PROGRAM F60_METS_Outputs
VAR
	//test : BOOL;
	fbForceOutputs					: FB_IO2_ForceOutputs;

	fbEUCAMachineRun_PulseGen		: FB_SquareWave;
	fbCaseContentOK_PulseGen		: FB_SquareWave;
	fbCaseValidationOK_PulseGen		: FB_SquareWave;
	fbOuterValidationOK_PulseGen	: FB_SquareWave;
	fbLabellerInhibit_PulseGen			: FB_SquareWave;
	fbTPDMachineRun_PulseGen		: FB_SquareWave;


	fbSafetyResetSignal				: FB_IO2_OutputCtrl;		(**)
	fbAdditionalSafetyResetSignal		: FB_IO2_OutputCtrl;
	fbResetPBIndicator					: FB_IO2_OutputCtrl;

	tofTPDMachineRunOff				: TOF;
	tofEUCAPreMachineRunOff			: TOF;
	tofEUCAMachineRunOff			: TOF;

	fbTPDMachineRun				: FB_IO2_OutputCtrl;
	fbCMLConvoyerRun			: FB_IO2_OutputCtrl;
	fbEUCAPreMachineRun			: FB_IO2_OutputCtrl;
	fbEUCAMachineRun			: FB_IO2_OutputCtrl;

	fbCaseContentOK				: FB_IO2_OutputCtrl;
	fbCaseValidationOK			: FB_IO2_OutputCtrl;
	fbOuterValidationOK			: FB_IO2_OutputCtrl;
	fbLabellerInhibit				: FB_IO2_OutputCtrl;

	ftrigPrintWhiteLable			: F_TRIG;

	fbPackAggregCamLensAir		: FB_IO2_OutputCtrl;
	fbOuterAggregCamLensAir	: FB_IO2_OutputCtrl;

	(*fbMLCameraLightning			: FB_IO2_OutputCtrl;
	fbAggCameraLightning		: FB_IO2_OutputCtrl;
	fbConfCameraLightning		: FB_IO2_OutputCtrl;
	fbOuterAggCameraLightning	: FB_IO2_OutputCtrl;*

	fbCamera01Lightning				: FB_IO2_OutputCtrl;
	fbCamera02Lightning				: FB_IO2_OutputCtrl;
	fbCamera03Lightning				: FB_IO2_OutputCtrl;
	fbCamera04Lightning				: FB_IO2_OutputCtrl;
	fbCamera05Lightning				: FB_IO2_OutputCtrl;
	fbCamera06Lightning				: FB_IO2_OutputCtrl;
	fbCamera07Lightning				: FB_IO2_OutputCtrl;
	fbCamera08Lightning				: FB_IO2_OutputCtrl;
	fbCamera09Lightning				: FB_IO2_OutputCtrl;
	fbCamera10Lightning				: FB_IO2_OutputCtrl;
	fbCamera11Lightning				: FB_IO2_OutputCtrl;
	fbCamera12Lightning				: FB_IO2_OutputCtrl;*


	fbCamera01Out				: FB_IO2_OutputCtrl;
	fbCamera02Out				: FB_IO2_OutputCtrl;
	fbCamera03Out				: FB_IO2_OutputCtrl;
	fbCamera04Out				: FB_IO2_OutputCtrl;
	fbCamera05Out				: FB_IO2_OutputCtrl;
	fbCamera06Out				: FB_IO2_OutputCtrl;
	fbCamera07Out				: FB_IO2_OutputCtrl;
	fbCamera08Out				: FB_IO2_OutputCtrl;
	fbCamera09Out				: FB_IO2_OutputCtrl;
	fbCamera10Out				: FB_IO2_OutputCtrl;
	fbCamera11Out				: FB_IO2_OutputCtrl;
	fbCamera12Out				: FB_IO2_OutputCtrl;*)

	aCameraOutControl			: ARRAY[1..cMAX_CAMERA_NUMBER] OF FB_IO2_OutputCtrl;
	aCameraLightControl			: ARRAY[1..cMAX_CAMERA_NUMBER] OF FB_IO2_OutputCtrl;

	fbLightPoleGreen				: FB_IO2_OutputCtrl;
	fbbLightPoleAmber			: FB_IO2_OutputCtrl;
	fbLightPoleRed					: FB_IO2_OutputCtrl;
	fbLightPoleAlarm				: FB_IO2_OutputCtrl;
	fbHandScannerGreen			: FB_IO2_OutputCtrl;
	fbHandScannerRed				: FB_IO2_OutputCtrl;
	fbGreenButtonLamp			: FB_IO2_OutputCtrl;

	fbDriveFaultAcknowledge		: FB_IO2_OutputCtrl;
	fbSideBeltDriveBrake			: FB_IO2_OutputCtrl;
	fbInfeedConveyorDriveRun	: FB_IO2_OutputCtrl;
	fbPackSeparatorDriveBrake	: FB_IO2_OutputCtrl;
	fbPackSeparationDriveRun		: FB_IO2_OutputCtrl;

	fbAdditionalConveyor1Run	: FB_IO2_OutputCtrl;
	fbAdditionalConveyor2Run	: FB_IO2_OutputCtrl;
	fbAdditionalConveyor3Run	: FB_IO2_OutputCtrl;
	fbAdditionalConveyor4Run	: FB_IO2_OutputCtrl;

	fbClampCylinderExtend		: FB_IO2_OutputCtrl;
	fbClampCylinderRetract		: FB_IO2_OutputCtrl;
	fbGateCylinderExtend			: FB_IO2_OutputCtrl;
	fbGateCylinderRetract			: FB_IO2_OutputCtrl;
	fbRejectCylinderExtend		: FB_IO2_OutputCtrl;
	fbRejectCylinderRetract		: FB_IO2_OutputCtrl;
	fbAdditionalRejectCylinderExtend		: FB_IO2_OutputCtrl;
	fbAdditionalRejectCylinderRetract		: FB_IO2_OutputCtrl;
	fbFirstPusherCylinderExtend		: FB_IO2_OutputCtrl;
	fbFirstPusherCylinderRetract		: FB_IO2_OutputCtrl;
	fbSecondPusherCylinderExtend		: FB_IO2_OutputCtrl;
	fbSecondPusherCylinderRetract		: FB_IO2_OutputCtrl;
	fbRejectActiveNCW				: FB_IO2_OutputCtrl;

	fbLaserEnable					: FB_IO2_OutputCtrl;
	fbLaserPrintAllow				: FB_IO2_OutputCtrl;
	fbLaserPrintStart				: FB_IO2_OutputCtrl;

	fbLabeller1Reset				: FB_IO2_OutputCtrl;
	fbLabeller1Print				: FB_IO2_OutputCtrl;
	fbWhiteLabe11Print			: FB_IO2_OutputCtrl;
	fbLabeller1Apply				: FB_IO2_OutputCtrl;
	fbLabbeller1ApplyAvailable	: FB_IO2_OutputCtrl;

	fbLabeller2Reset				: FB_IO2_OutputCtrl;
	fbLabeller2Print				: FB_IO2_OutputCtrl;
	fbWhiteLabe12Print			: FB_IO2_OutputCtrl;
	fbLabeller2Apply				: FB_IO2_OutputCtrl;
	fbLabbeller2ApplyAvailable	: FB_IO2_OutputCtrl;

	fbIntermediatePrinterTrigger1	: FB_IO2_OutputCtrl;

	bDummyOutput				: BOOL;
	nDummyOutput				: INT;

END_VAR
VAR // added by the converter: edge detectors and wires of the graphical bodies
    _w1 : BOOL;
END_VAR

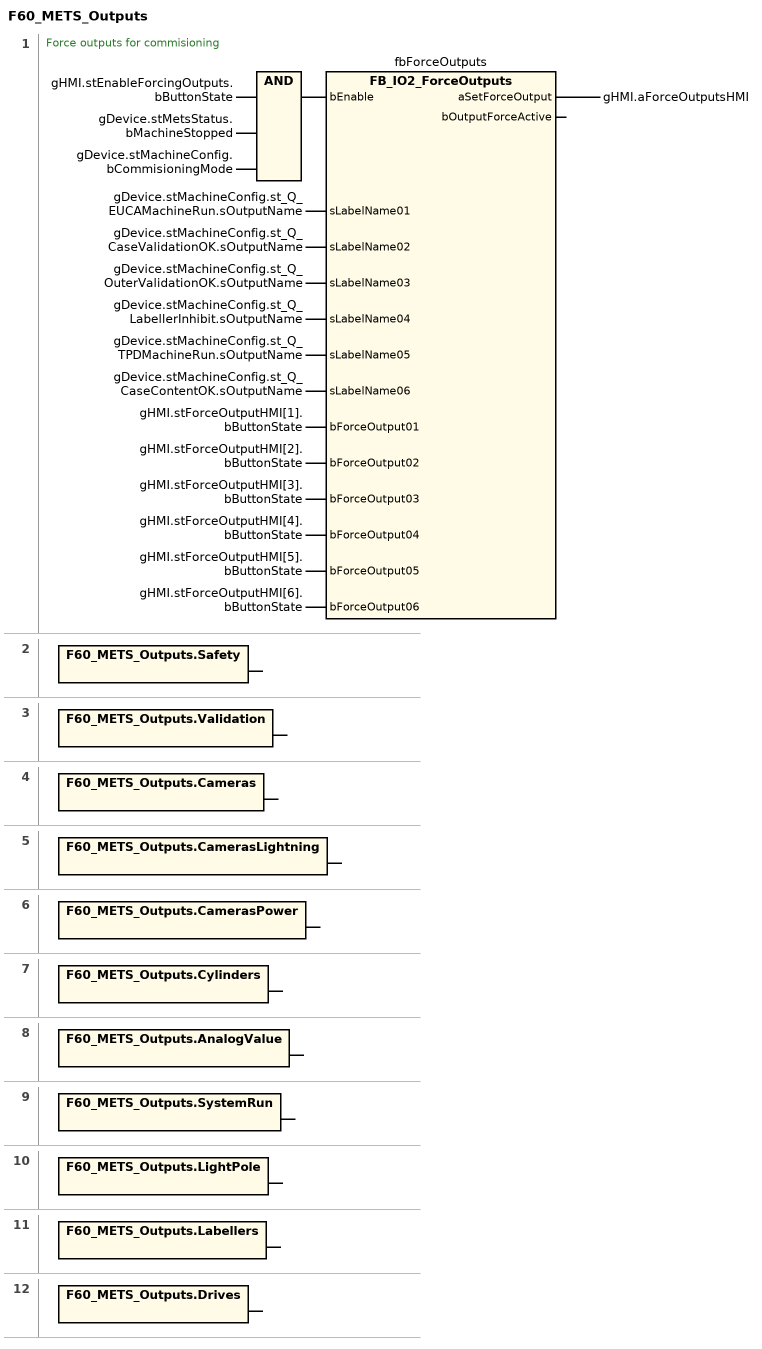
// NETWORK 1
// Force outputs for commisioning
fbForceOutputs(
    bEnable := gHMI.stEnableForcingOutputs.bButtonState AND gDevice.stMetsStatus.bMachineStopped AND gDevice.stMachineConfig.bCommisioningMode,
    sLabelName01 := gDevice.stMachineConfig.st_Q_EUCAMachineRun.sOutputName,
    sLabelName02 := gDevice.stMachineConfig.st_Q_CaseValidationOK.sOutputName,
    sLabelName03 := gDevice.stMachineConfig.st_Q_OuterValidationOK.sOutputName,
    sLabelName04 := gDevice.stMachineConfig.st_Q_LabellerInhibit.sOutputName,
    sLabelName05 := gDevice.stMachineConfig.st_Q_TPDMachineRun.sOutputName,
    sLabelName06 := gDevice.stMachineConfig.st_Q_CaseContentOK.sOutputName,
    bForceOutput01 := gHMI.stForceOutputHMI[1].bButtonState,
    bForceOutput02 := gHMI.stForceOutputHMI[2].bButtonState,
    bForceOutput03 := gHMI.stForceOutputHMI[3].bButtonState,
    bForceOutput04 := gHMI.stForceOutputHMI[4].bButtonState,
    bForceOutput05 := gHMI.stForceOutputHMI[5].bButtonState,
    bForceOutput06 := gHMI.stForceOutputHMI[6].bButtonState); // FB_IO2_ForceOutputs
gHMI.aForceOutputsHMI := fbForceOutputs.aSetForceOutput;

// NETWORK 2
F60_METS_Outputs.Safety();

// NETWORK 3
F60_METS_Outputs.Validation();

// NETWORK 4
F60_METS_Outputs.Cameras();

// NETWORK 5
F60_METS_Outputs.CamerasLightning();

// NETWORK 6
F60_METS_Outputs.CamerasPower();

// NETWORK 7
F60_METS_Outputs.Cylinders();

// NETWORK 8
F60_METS_Outputs.AnalogValue();

// NETWORK 9
F60_METS_Outputs.SystemRun();

// NETWORK 10
F60_METS_Outputs.LightPole();

// NETWORK 11
F60_METS_Outputs.Labellers();

// NETWORK 12
F60_METS_Outputs.Drives();

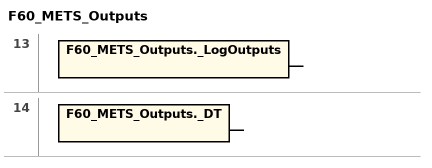
// NETWORK 13
F60_METS_Outputs._LogOutputs();

// NETWORK 14
F60_METS_Outputs._DT();

ACTION _DT:
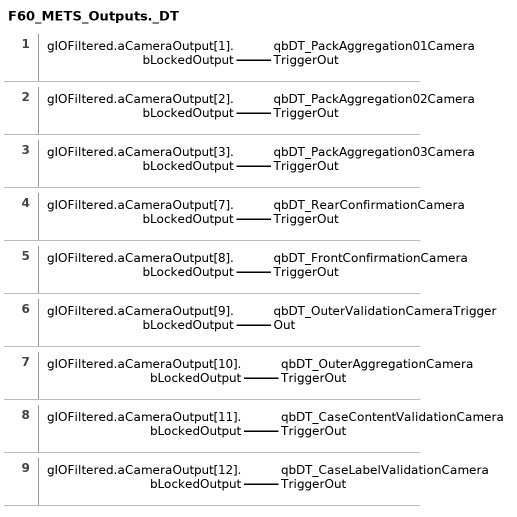
// NETWORK 1
qbDT_PackAggregation01CameraTriggerOut := gIOFiltered.aCameraOutput[1].bLockedOutput;

// NETWORK 2
qbDT_PackAggregation02CameraTriggerOut := gIOFiltered.aCameraOutput[2].bLockedOutput;

// NETWORK 3
qbDT_PackAggregation03CameraTriggerOut := gIOFiltered.aCameraOutput[3].bLockedOutput;

// NETWORK 4
qbDT_RearConfirmationCameraTriggerOut := gIOFiltered.aCameraOutput[7].bLockedOutput;

// NETWORK 5
qbDT_FrontConfirmationCameraTriggerOut := gIOFiltered.aCameraOutput[8].bLockedOutput;

// NETWORK 6
qbDT_OuterValidationCameraTriggerOut := gIOFiltered.aCameraOutput[9].bLockedOutput;

// NETWORK 7
qbDT_OuterAggregationCameraTriggerOut := gIOFiltered.aCameraOutput[10].bLockedOutput;

// NETWORK 8
qbDT_CaseContentValidationCameraTriggerOut := gIOFiltered.aCameraOutput[11].bLockedOutput;

// NETWORK 9
qbDT_CaseLabelValidationCameraTriggerOut := gIOFiltered.aCameraOutput[12].bLockedOutput;
END_ACTION

ACTION _LogOutputs:
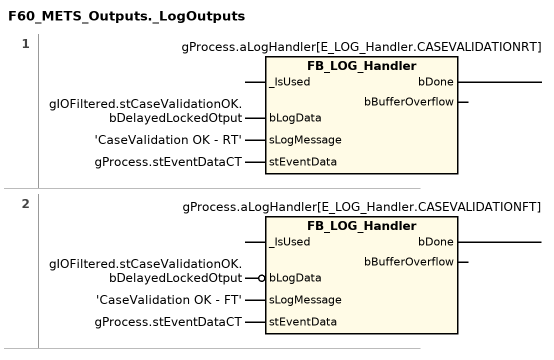
// NETWORK 1
gProcess.aLogHandler[E_LOG_Handler.CASEVALIDATIONRT](
    bLogData := gIOFiltered.stCaseValidationOK.bDelayedLockedOtput,
    sLogMessage := 'CaseValidation OK - RT',
    stEventData := gProcess.stEventDataCT); // FB_LOG_Handler

// NETWORK 2
gProcess.aLogHandler[E_LOG_Handler.CASEVALIDATIONFT](
    bLogData := NOT gIOFiltered.stCaseValidationOK.bDelayedLockedOtput,
    sLogMessage := 'CaseValidation OK - FT',
    stEventData := gProcess.stEventDataCT); // FB_LOG_Handler
END_ACTION

ACTION AnalogValue:
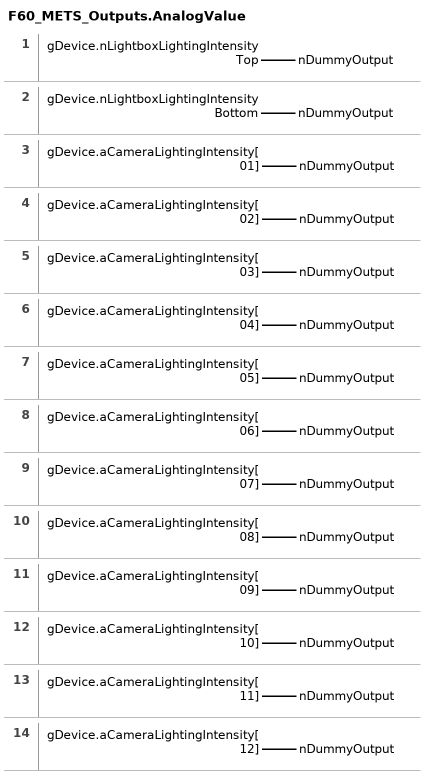
// NETWORK 1
nDummyOutput := gDevice.nLightboxLightingIntensityTop;

// NETWORK 2
nDummyOutput := gDevice.nLightboxLightingIntensityBottom;

// NETWORK 3
nDummyOutput := gDevice.aCameraLightingIntensity[01];

// NETWORK 4
nDummyOutput := gDevice.aCameraLightingIntensity[02];

// NETWORK 5
nDummyOutput := gDevice.aCameraLightingIntensity[03];

// NETWORK 6
nDummyOutput := gDevice.aCameraLightingIntensity[04];

// NETWORK 7
nDummyOutput := gDevice.aCameraLightingIntensity[05];

// NETWORK 8
nDummyOutput := gDevice.aCameraLightingIntensity[06];

// NETWORK 9
nDummyOutput := gDevice.aCameraLightingIntensity[07];

// NETWORK 10
nDummyOutput := gDevice.aCameraLightingIntensity[08];

// NETWORK 11
nDummyOutput := gDevice.aCameraLightingIntensity[09];

// NETWORK 12
nDummyOutput := gDevice.aCameraLightingIntensity[10];

// NETWORK 13
nDummyOutput := gDevice.aCameraLightingIntensity[11];

// NETWORK 14
nDummyOutput := gDevice.aCameraLightingIntensity[12];
END_ACTION

ACTION Cameras:
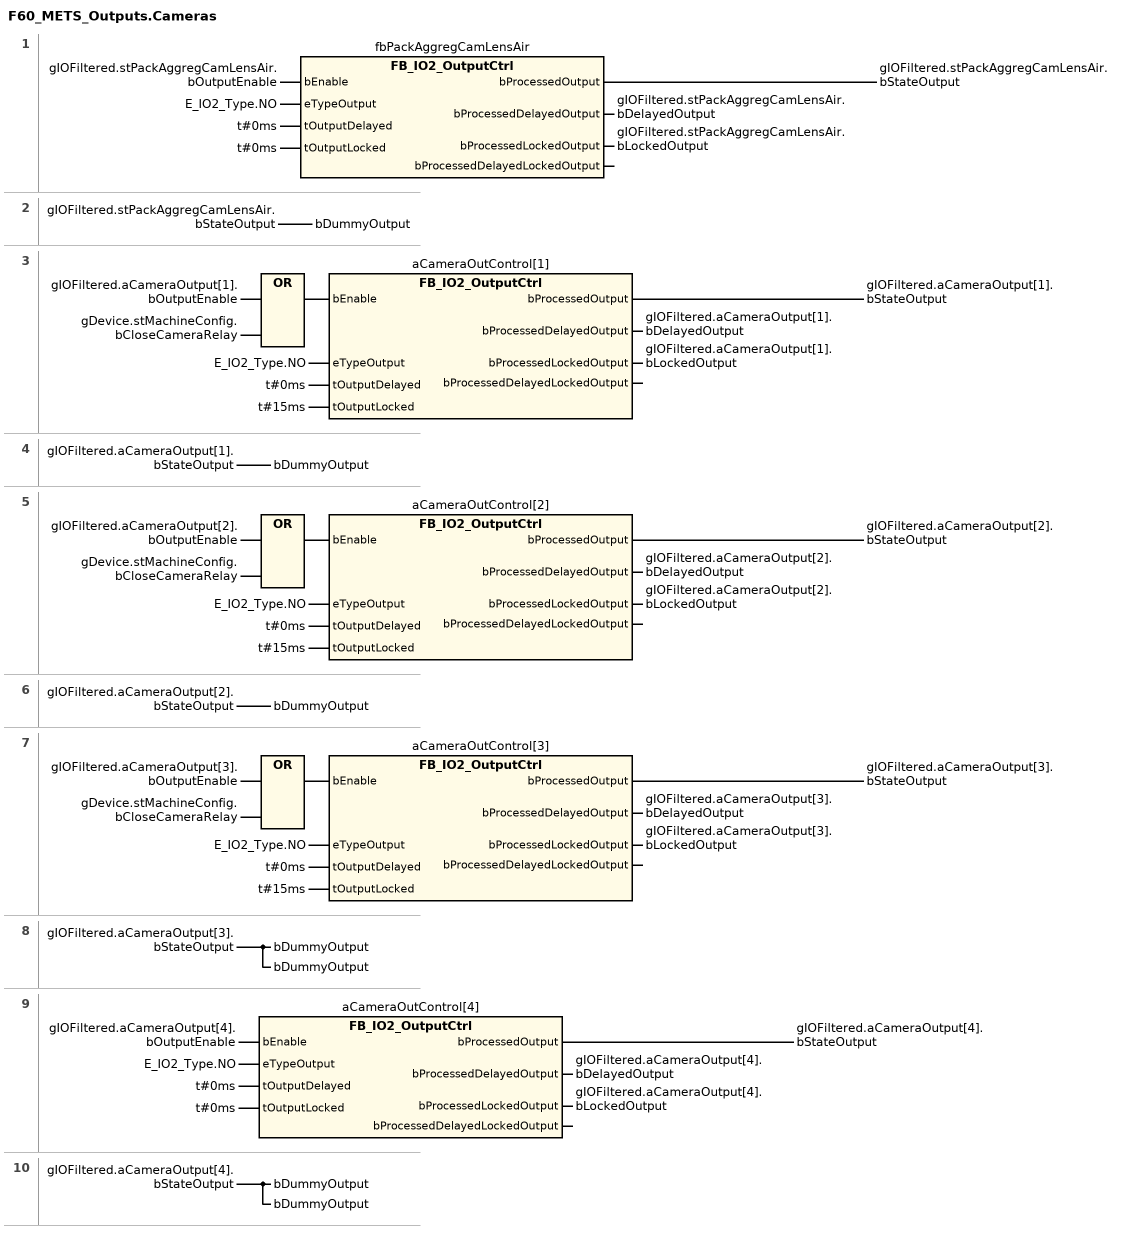
// NETWORK 1
fbPackAggregCamLensAir(
    bEnable := gIOFiltered.stPackAggregCamLensAir.bOutputEnable,
    eTypeOutput := E_IO2_Type.NO,
    tOutputDelayed := t#0ms,
    tOutputLocked := t#0ms,
    bProcessedDelayedOutput => gIOFiltered.stPackAggregCamLensAir.bDelayedOutput,
    bProcessedLockedOutput => gIOFiltered.stPackAggregCamLensAir.bLockedOutput); // FB_IO2_OutputCtrl
gIOFiltered.stPackAggregCamLensAir.bStateOutput := fbPackAggregCamLensAir.bProcessedOutput;

// NETWORK 2
bDummyOutput := gIOFiltered.stPackAggregCamLensAir.bStateOutput;

// NETWORK 3
aCameraOutControl[1](
    bEnable := gIOFiltered.aCameraOutput[1].bOutputEnable OR gDevice.stMachineConfig.bCloseCameraRelay,
    eTypeOutput := E_IO2_Type.NO,
    tOutputDelayed := t#0ms,
    tOutputLocked := t#15ms,
    bProcessedDelayedOutput => gIOFiltered.aCameraOutput[1].bDelayedOutput,
    bProcessedLockedOutput => gIOFiltered.aCameraOutput[1].bLockedOutput); // FB_IO2_OutputCtrl
gIOFiltered.aCameraOutput[1].bStateOutput := aCameraOutControl[1].bProcessedOutput;

// NETWORK 4
bDummyOutput := gIOFiltered.aCameraOutput[1].bStateOutput;

// NETWORK 5
aCameraOutControl[2](
    bEnable := gIOFiltered.aCameraOutput[2].bOutputEnable OR gDevice.stMachineConfig.bCloseCameraRelay,
    eTypeOutput := E_IO2_Type.NO,
    tOutputDelayed := t#0ms,
    tOutputLocked := t#15ms,
    bProcessedDelayedOutput => gIOFiltered.aCameraOutput[2].bDelayedOutput,
    bProcessedLockedOutput => gIOFiltered.aCameraOutput[2].bLockedOutput); // FB_IO2_OutputCtrl
gIOFiltered.aCameraOutput[2].bStateOutput := aCameraOutControl[2].bProcessedOutput;

// NETWORK 6
bDummyOutput := gIOFiltered.aCameraOutput[2].bStateOutput;

// NETWORK 7
aCameraOutControl[3](
    bEnable := gIOFiltered.aCameraOutput[3].bOutputEnable OR gDevice.stMachineConfig.bCloseCameraRelay,
    eTypeOutput := E_IO2_Type.NO,
    tOutputDelayed := t#0ms,
    tOutputLocked := t#15ms,
    bProcessedDelayedOutput => gIOFiltered.aCameraOutput[3].bDelayedOutput,
    bProcessedLockedOutput => gIOFiltered.aCameraOutput[3].bLockedOutput); // FB_IO2_OutputCtrl
gIOFiltered.aCameraOutput[3].bStateOutput := aCameraOutControl[3].bProcessedOutput;

// NETWORK 8
bDummyOutput := gIOFiltered.aCameraOutput[3].bStateOutput;
bDummyOutput := gIOFiltered.aCameraOutput[3].bStateOutput;

// NETWORK 9
aCameraOutControl[4](
    bEnable := gIOFiltered.aCameraOutput[4].bOutputEnable,
    eTypeOutput := E_IO2_Type.NO,
    tOutputDelayed := t#0ms,
    tOutputLocked := t#0ms,
    bProcessedDelayedOutput => gIOFiltered.aCameraOutput[4].bDelayedOutput,
    bProcessedLockedOutput => gIOFiltered.aCameraOutput[4].bLockedOutput); // FB_IO2_OutputCtrl
gIOFiltered.aCameraOutput[4].bStateOutput := aCameraOutControl[4].bProcessedOutput;

// NETWORK 10
bDummyOutput := gIOFiltered.aCameraOutput[4].bStateOutput;
bDummyOutput := gIOFiltered.aCameraOutput[4].bStateOutput;

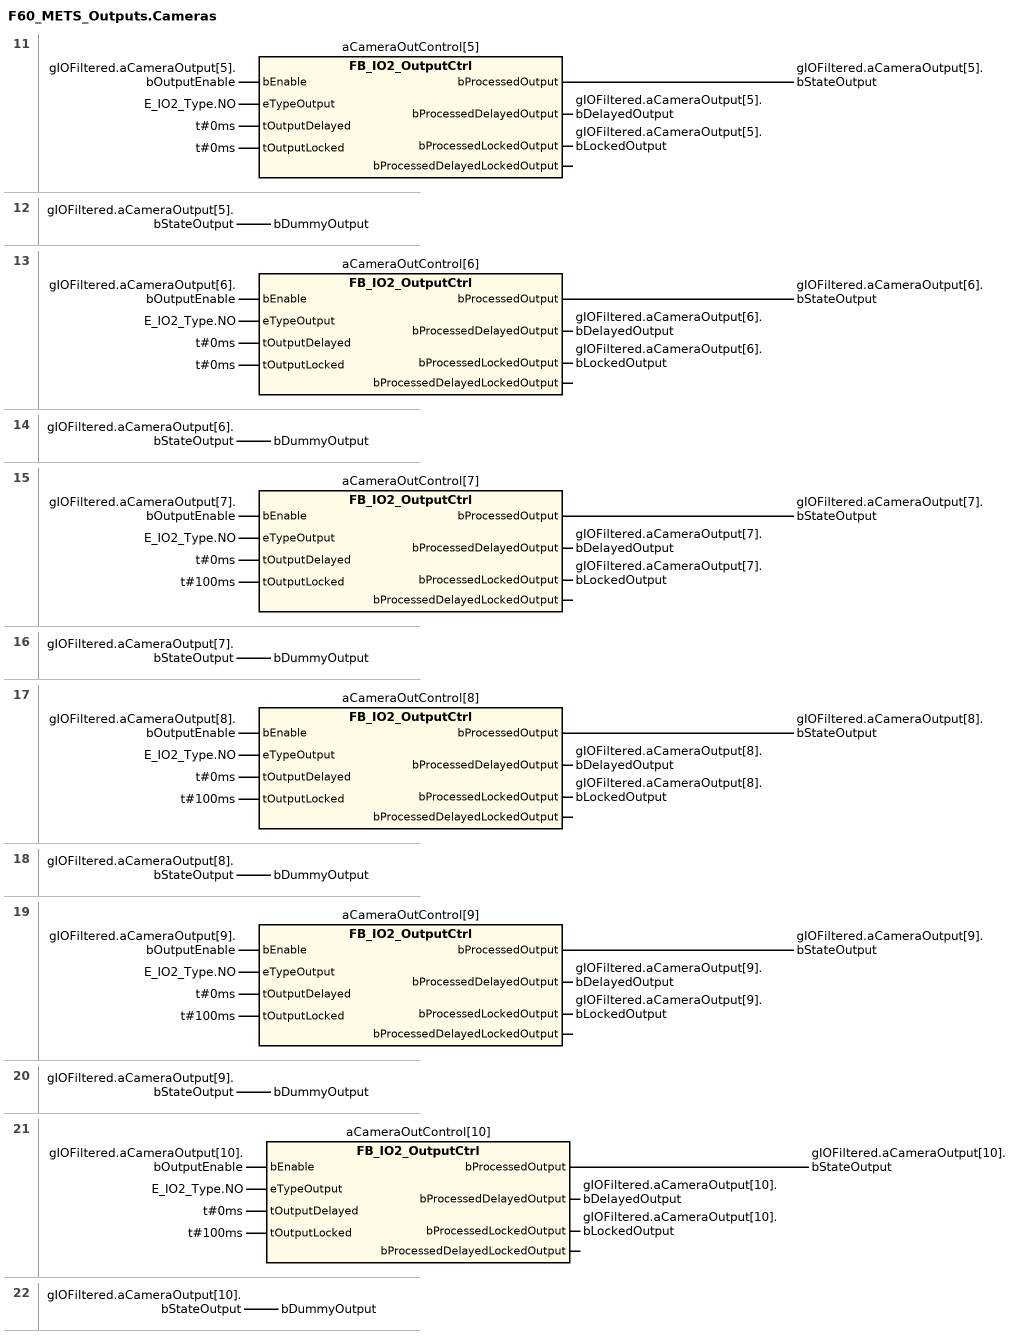
// NETWORK 11
aCameraOutControl[5](
    bEnable := gIOFiltered.aCameraOutput[5].bOutputEnable,
    eTypeOutput := E_IO2_Type.NO,
    tOutputDelayed := t#0ms,
    tOutputLocked := t#0ms,
    bProcessedDelayedOutput => gIOFiltered.aCameraOutput[5].bDelayedOutput,
    bProcessedLockedOutput => gIOFiltered.aCameraOutput[5].bLockedOutput); // FB_IO2_OutputCtrl
gIOFiltered.aCameraOutput[5].bStateOutput := aCameraOutControl[5].bProcessedOutput;

// NETWORK 12
bDummyOutput := gIOFiltered.aCameraOutput[5].bStateOutput;

// NETWORK 13
aCameraOutControl[6](
    bEnable := gIOFiltered.aCameraOutput[6].bOutputEnable,
    eTypeOutput := E_IO2_Type.NO,
    tOutputDelayed := t#0ms,
    tOutputLocked := t#0ms,
    bProcessedDelayedOutput => gIOFiltered.aCameraOutput[6].bDelayedOutput,
    bProcessedLockedOutput => gIOFiltered.aCameraOutput[6].bLockedOutput); // FB_IO2_OutputCtrl
gIOFiltered.aCameraOutput[6].bStateOutput := aCameraOutControl[6].bProcessedOutput;

// NETWORK 14
bDummyOutput := gIOFiltered.aCameraOutput[6].bStateOutput;

// NETWORK 15
aCameraOutControl[7](
    bEnable := gIOFiltered.aCameraOutput[7].bOutputEnable,
    eTypeOutput := E_IO2_Type.NO,
    tOutputDelayed := t#0ms,
    tOutputLocked := t#100ms,
    bProcessedDelayedOutput => gIOFiltered.aCameraOutput[7].bDelayedOutput,
    bProcessedLockedOutput => gIOFiltered.aCameraOutput[7].bLockedOutput); // FB_IO2_OutputCtrl
gIOFiltered.aCameraOutput[7].bStateOutput := aCameraOutControl[7].bProcessedOutput;

// NETWORK 16
bDummyOutput := gIOFiltered.aCameraOutput[7].bStateOutput;

// NETWORK 17
aCameraOutControl[8](
    bEnable := gIOFiltered.aCameraOutput[8].bOutputEnable,
    eTypeOutput := E_IO2_Type.NO,
    tOutputDelayed := t#0ms,
    tOutputLocked := t#100ms,
    bProcessedDelayedOutput => gIOFiltered.aCameraOutput[8].bDelayedOutput,
    bProcessedLockedOutput => gIOFiltered.aCameraOutput[8].bLockedOutput); // FB_IO2_OutputCtrl
gIOFiltered.aCameraOutput[8].bStateOutput := aCameraOutControl[8].bProcessedOutput;

// NETWORK 18
bDummyOutput := gIOFiltered.aCameraOutput[8].bStateOutput;

// NETWORK 19
aCameraOutControl[9](
    bEnable := gIOFiltered.aCameraOutput[9].bOutputEnable,
    eTypeOutput := E_IO2_Type.NO,
    tOutputDelayed := t#0ms,
    tOutputLocked := t#100ms,
    bProcessedDelayedOutput => gIOFiltered.aCameraOutput[9].bDelayedOutput,
    bProcessedLockedOutput => gIOFiltered.aCameraOutput[9].bLockedOutput); // FB_IO2_OutputCtrl
gIOFiltered.aCameraOutput[9].bStateOutput := aCameraOutControl[9].bProcessedOutput;

// NETWORK 20
bDummyOutput := gIOFiltered.aCameraOutput[9].bStateOutput;

// NETWORK 21
aCameraOutControl[10](
    bEnable := gIOFiltered.aCameraOutput[10].bOutputEnable,
    eTypeOutput := E_IO2_Type.NO,
    tOutputDelayed := t#0ms,
    tOutputLocked := t#100ms,
    bProcessedDelayedOutput => gIOFiltered.aCameraOutput[10].bDelayedOutput,
    bProcessedLockedOutput => gIOFiltered.aCameraOutput[10].bLockedOutput); // FB_IO2_OutputCtrl
gIOFiltered.aCameraOutput[10].bStateOutput := aCameraOutControl[10].bProcessedOutput;

// NETWORK 22
bDummyOutput := gIOFiltered.aCameraOutput[10].bStateOutput;

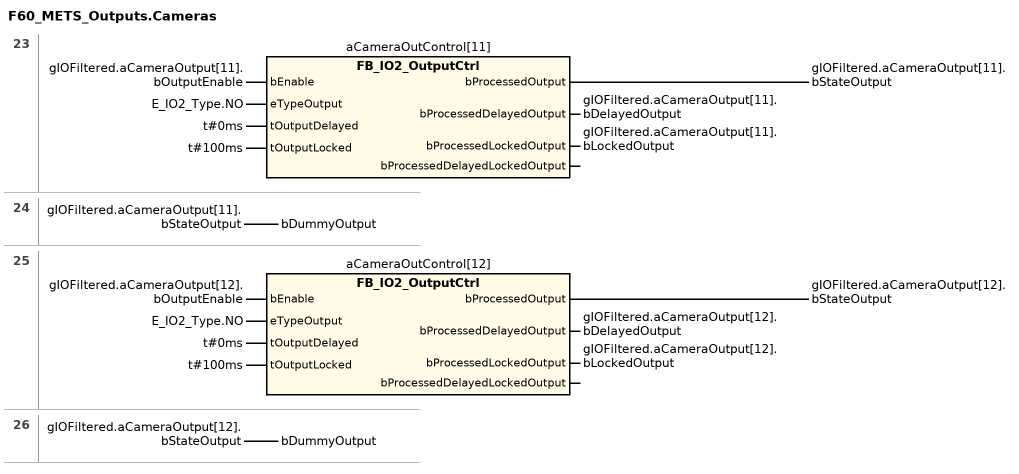
// NETWORK 23
aCameraOutControl[11](
    bEnable := gIOFiltered.aCameraOutput[11].bOutputEnable,
    eTypeOutput := E_IO2_Type.NO,
    tOutputDelayed := t#0ms,
    tOutputLocked := t#100ms,
    bProcessedDelayedOutput => gIOFiltered.aCameraOutput[11].bDelayedOutput,
    bProcessedLockedOutput => gIOFiltered.aCameraOutput[11].bLockedOutput); // FB_IO2_OutputCtrl
gIOFiltered.aCameraOutput[11].bStateOutput := aCameraOutControl[11].bProcessedOutput;

// NETWORK 24
bDummyOutput := gIOFiltered.aCameraOutput[11].bStateOutput;

// NETWORK 25
aCameraOutControl[12](
    bEnable := gIOFiltered.aCameraOutput[12].bOutputEnable,
    eTypeOutput := E_IO2_Type.NO,
    tOutputDelayed := t#0ms,
    tOutputLocked := t#100ms,
    bProcessedDelayedOutput => gIOFiltered.aCameraOutput[12].bDelayedOutput,
    bProcessedLockedOutput => gIOFiltered.aCameraOutput[12].bLockedOutput); // FB_IO2_OutputCtrl
gIOFiltered.aCameraOutput[12].bStateOutput := aCameraOutControl[12].bProcessedOutput;

// NETWORK 26
bDummyOutput := gIOFiltered.aCameraOutput[12].bStateOutput;
END_ACTION

ACTION CamerasLightning:
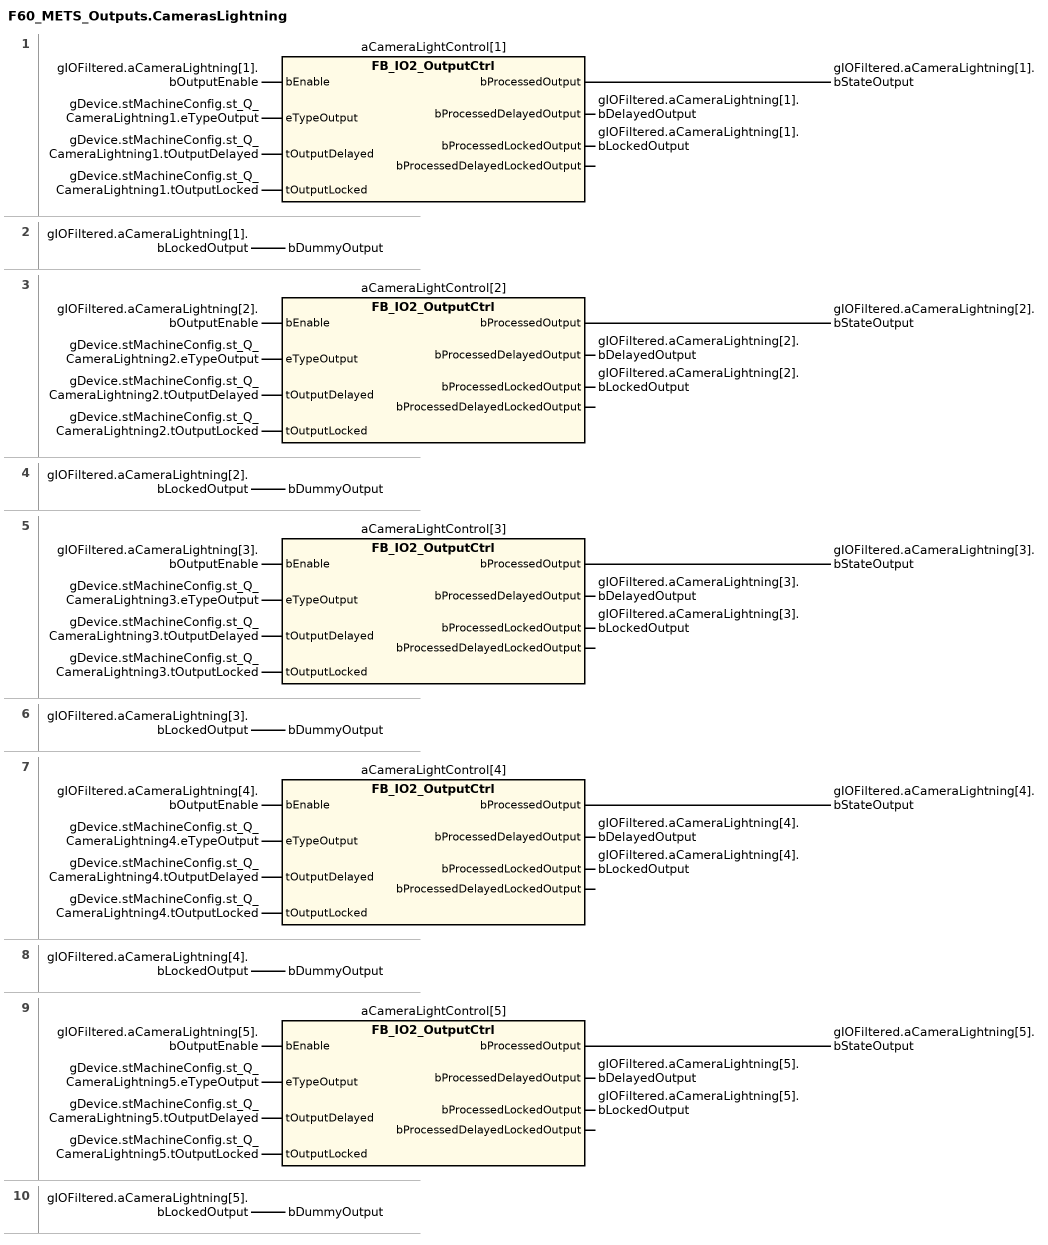
// NETWORK 1
aCameraLightControl[1](
    bEnable := gIOFiltered.aCameraLightning[1].bOutputEnable,
    eTypeOutput := gDevice.stMachineConfig.st_Q_CameraLightning1.eTypeOutput,
    tOutputDelayed := gDevice.stMachineConfig.st_Q_CameraLightning1.tOutputDelayed,
    tOutputLocked := gDevice.stMachineConfig.st_Q_CameraLightning1.tOutputLocked,
    bProcessedDelayedOutput => gIOFiltered.aCameraLightning[1].bDelayedOutput,
    bProcessedLockedOutput => gIOFiltered.aCameraLightning[1].bLockedOutput); // FB_IO2_OutputCtrl
gIOFiltered.aCameraLightning[1].bStateOutput := aCameraLightControl[1].bProcessedOutput;

// NETWORK 2
bDummyOutput := gIOFiltered.aCameraLightning[1].bLockedOutput;

// NETWORK 3
aCameraLightControl[2](
    bEnable := gIOFiltered.aCameraLightning[2].bOutputEnable,
    eTypeOutput := gDevice.stMachineConfig.st_Q_CameraLightning2.eTypeOutput,
    tOutputDelayed := gDevice.stMachineConfig.st_Q_CameraLightning2.tOutputDelayed,
    tOutputLocked := gDevice.stMachineConfig.st_Q_CameraLightning2.tOutputLocked,
    bProcessedDelayedOutput => gIOFiltered.aCameraLightning[2].bDelayedOutput,
    bProcessedLockedOutput => gIOFiltered.aCameraLightning[2].bLockedOutput); // FB_IO2_OutputCtrl
gIOFiltered.aCameraLightning[2].bStateOutput := aCameraLightControl[2].bProcessedOutput;

// NETWORK 4
bDummyOutput := gIOFiltered.aCameraLightning[2].bLockedOutput;

// NETWORK 5
aCameraLightControl[3](
    bEnable := gIOFiltered.aCameraLightning[3].bOutputEnable,
    eTypeOutput := gDevice.stMachineConfig.st_Q_CameraLightning3.eTypeOutput,
    tOutputDelayed := gDevice.stMachineConfig.st_Q_CameraLightning3.tOutputDelayed,
    tOutputLocked := gDevice.stMachineConfig.st_Q_CameraLightning3.tOutputLocked,
    bProcessedDelayedOutput => gIOFiltered.aCameraLightning[3].bDelayedOutput,
    bProcessedLockedOutput => gIOFiltered.aCameraLightning[3].bLockedOutput); // FB_IO2_OutputCtrl
gIOFiltered.aCameraLightning[3].bStateOutput := aCameraLightControl[3].bProcessedOutput;

// NETWORK 6
bDummyOutput := gIOFiltered.aCameraLightning[3].bLockedOutput;

// NETWORK 7
aCameraLightControl[4](
    bEnable := gIOFiltered.aCameraLightning[4].bOutputEnable,
    eTypeOutput := gDevice.stMachineConfig.st_Q_CameraLightning4.eTypeOutput,
    tOutputDelayed := gDevice.stMachineConfig.st_Q_CameraLightning4.tOutputDelayed,
    tOutputLocked := gDevice.stMachineConfig.st_Q_CameraLightning4.tOutputLocked,
    bProcessedDelayedOutput => gIOFiltered.aCameraLightning[4].bDelayedOutput,
    bProcessedLockedOutput => gIOFiltered.aCameraLightning[4].bLockedOutput); // FB_IO2_OutputCtrl
gIOFiltered.aCameraLightning[4].bStateOutput := aCameraLightControl[4].bProcessedOutput;

// NETWORK 8
bDummyOutput := gIOFiltered.aCameraLightning[4].bLockedOutput;

// NETWORK 9
aCameraLightControl[5](
    bEnable := gIOFiltered.aCameraLightning[5].bOutputEnable,
    eTypeOutput := gDevice.stMachineConfig.st_Q_CameraLightning5.eTypeOutput,
    tOutputDelayed := gDevice.stMachineConfig.st_Q_CameraLightning5.tOutputDelayed,
    tOutputLocked := gDevice.stMachineConfig.st_Q_CameraLightning5.tOutputLocked,
    bProcessedDelayedOutput => gIOFiltered.aCameraLightning[5].bDelayedOutput,
    bProcessedLockedOutput => gIOFiltered.aCameraLightning[5].bLockedOutput); // FB_IO2_OutputCtrl
gIOFiltered.aCameraLightning[5].bStateOutput := aCameraLightControl[5].bProcessedOutput;

// NETWORK 10
bDummyOutput := gIOFiltered.aCameraLightning[5].bLockedOutput;

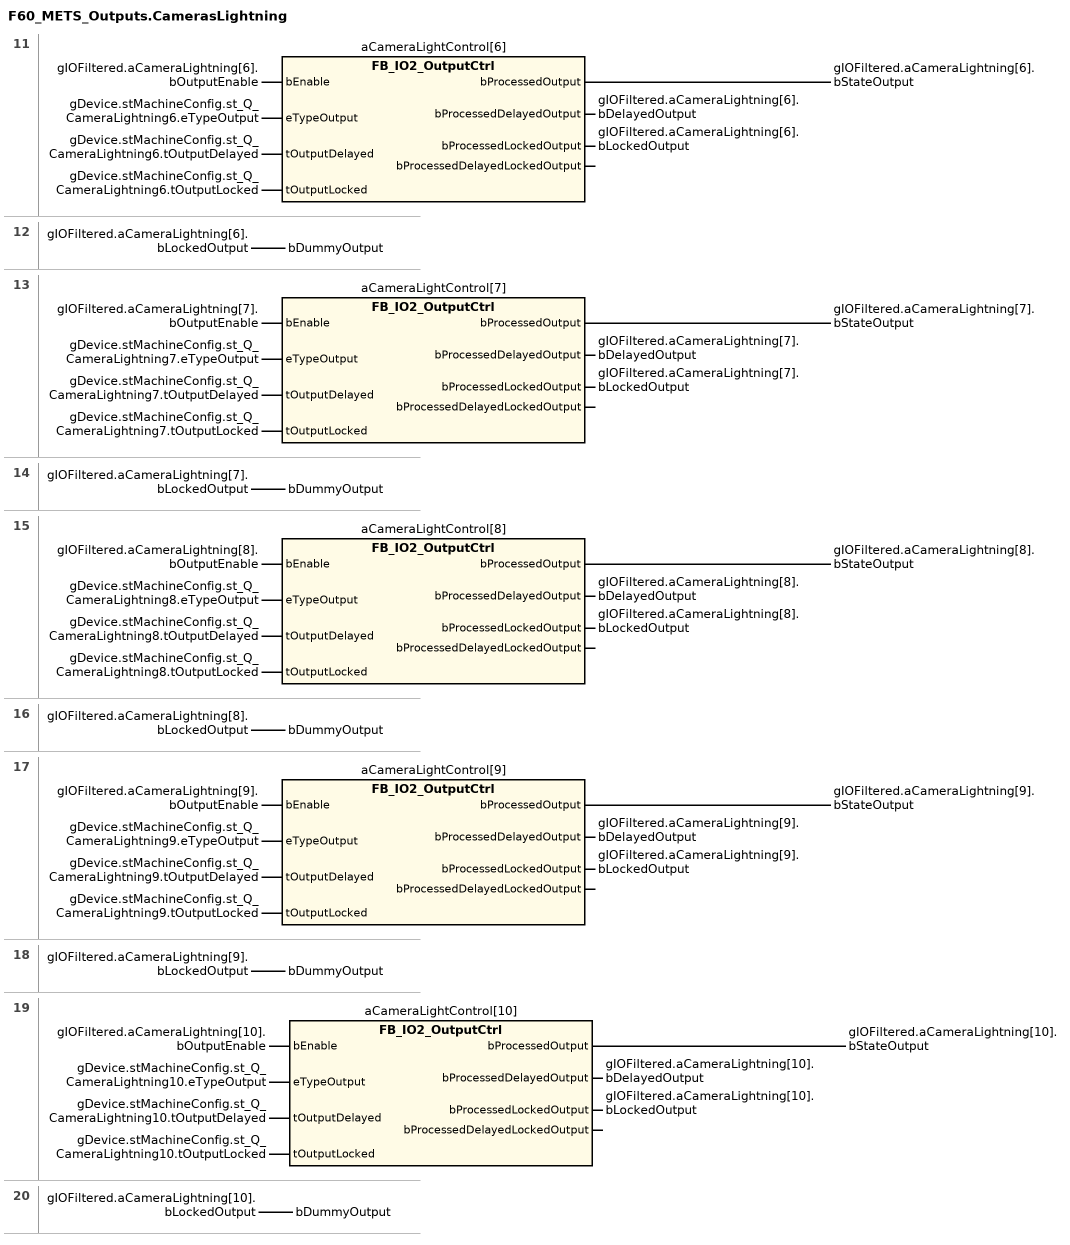
// NETWORK 11
aCameraLightControl[6](
    bEnable := gIOFiltered.aCameraLightning[6].bOutputEnable,
    eTypeOutput := gDevice.stMachineConfig.st_Q_CameraLightning6.eTypeOutput,
    tOutputDelayed := gDevice.stMachineConfig.st_Q_CameraLightning6.tOutputDelayed,
    tOutputLocked := gDevice.stMachineConfig.st_Q_CameraLightning6.tOutputLocked,
    bProcessedDelayedOutput => gIOFiltered.aCameraLightning[6].bDelayedOutput,
    bProcessedLockedOutput => gIOFiltered.aCameraLightning[6].bLockedOutput); // FB_IO2_OutputCtrl
gIOFiltered.aCameraLightning[6].bStateOutput := aCameraLightControl[6].bProcessedOutput;

// NETWORK 12
bDummyOutput := gIOFiltered.aCameraLightning[6].bLockedOutput;

// NETWORK 13
aCameraLightControl[7](
    bEnable := gIOFiltered.aCameraLightning[7].bOutputEnable,
    eTypeOutput := gDevice.stMachineConfig.st_Q_CameraLightning7.eTypeOutput,
    tOutputDelayed := gDevice.stMachineConfig.st_Q_CameraLightning7.tOutputDelayed,
    tOutputLocked := gDevice.stMachineConfig.st_Q_CameraLightning7.tOutputLocked,
    bProcessedDelayedOutput => gIOFiltered.aCameraLightning[7].bDelayedOutput,
    bProcessedLockedOutput => gIOFiltered.aCameraLightning[7].bLockedOutput); // FB_IO2_OutputCtrl
gIOFiltered.aCameraLightning[7].bStateOutput := aCameraLightControl[7].bProcessedOutput;

// NETWORK 14
bDummyOutput := gIOFiltered.aCameraLightning[7].bLockedOutput;

// NETWORK 15
aCameraLightControl[8](
    bEnable := gIOFiltered.aCameraLightning[8].bOutputEnable,
    eTypeOutput := gDevice.stMachineConfig.st_Q_CameraLightning8.eTypeOutput,
    tOutputDelayed := gDevice.stMachineConfig.st_Q_CameraLightning8.tOutputDelayed,
    tOutputLocked := gDevice.stMachineConfig.st_Q_CameraLightning8.tOutputLocked,
    bProcessedDelayedOutput => gIOFiltered.aCameraLightning[8].bDelayedOutput,
    bProcessedLockedOutput => gIOFiltered.aCameraLightning[8].bLockedOutput); // FB_IO2_OutputCtrl
gIOFiltered.aCameraLightning[8].bStateOutput := aCameraLightControl[8].bProcessedOutput;

// NETWORK 16
bDummyOutput := gIOFiltered.aCameraLightning[8].bLockedOutput;

// NETWORK 17
aCameraLightControl[9](
    bEnable := gIOFiltered.aCameraLightning[9].bOutputEnable,
    eTypeOutput := gDevice.stMachineConfig.st_Q_CameraLightning9.eTypeOutput,
    tOutputDelayed := gDevice.stMachineConfig.st_Q_CameraLightning9.tOutputDelayed,
    tOutputLocked := gDevice.stMachineConfig.st_Q_CameraLightning9.tOutputLocked,
    bProcessedDelayedOutput => gIOFiltered.aCameraLightning[9].bDelayedOutput,
    bProcessedLockedOutput => gIOFiltered.aCameraLightning[9].bLockedOutput); // FB_IO2_OutputCtrl
gIOFiltered.aCameraLightning[9].bStateOutput := aCameraLightControl[9].bProcessedOutput;

// NETWORK 18
bDummyOutput := gIOFiltered.aCameraLightning[9].bLockedOutput;

// NETWORK 19
aCameraLightControl[10](
    bEnable := gIOFiltered.aCameraLightning[10].bOutputEnable,
    eTypeOutput := gDevice.stMachineConfig.st_Q_CameraLightning10.eTypeOutput,
    tOutputDelayed := gDevice.stMachineConfig.st_Q_CameraLightning10.tOutputDelayed,
    tOutputLocked := gDevice.stMachineConfig.st_Q_CameraLightning10.tOutputLocked,
    bProcessedDelayedOutput => gIOFiltered.aCameraLightning[10].bDelayedOutput,
    bProcessedLockedOutput => gIOFiltered.aCameraLightning[10].bLockedOutput); // FB_IO2_OutputCtrl
gIOFiltered.aCameraLightning[10].bStateOutput := aCameraLightControl[10].bProcessedOutput;

// NETWORK 20
bDummyOutput := gIOFiltered.aCameraLightning[10].bLockedOutput;

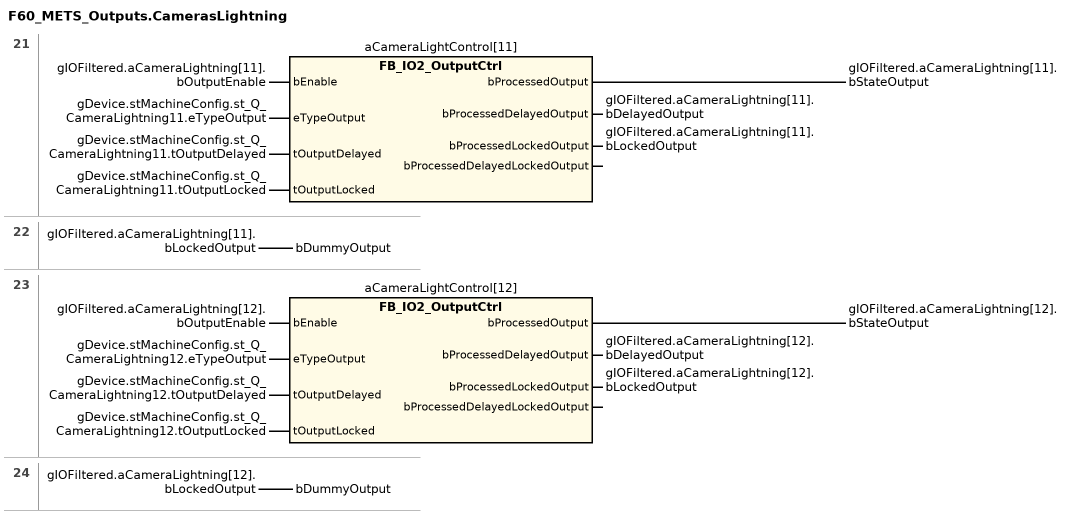
// NETWORK 21
aCameraLightControl[11](
    bEnable := gIOFiltered.aCameraLightning[11].bOutputEnable,
    eTypeOutput := gDevice.stMachineConfig.st_Q_CameraLightning11.eTypeOutput,
    tOutputDelayed := gDevice.stMachineConfig.st_Q_CameraLightning11.tOutputDelayed,
    tOutputLocked := gDevice.stMachineConfig.st_Q_CameraLightning11.tOutputLocked,
    bProcessedDelayedOutput => gIOFiltered.aCameraLightning[11].bDelayedOutput,
    bProcessedLockedOutput => gIOFiltered.aCameraLightning[11].bLockedOutput); // FB_IO2_OutputCtrl
gIOFiltered.aCameraLightning[11].bStateOutput := aCameraLightControl[11].bProcessedOutput;

// NETWORK 22
bDummyOutput := gIOFiltered.aCameraLightning[11].bLockedOutput;

// NETWORK 23
aCameraLightControl[12](
    bEnable := gIOFiltered.aCameraLightning[12].bOutputEnable,
    eTypeOutput := gDevice.stMachineConfig.st_Q_CameraLightning12.eTypeOutput,
    tOutputDelayed := gDevice.stMachineConfig.st_Q_CameraLightning12.tOutputDelayed,
    tOutputLocked := gDevice.stMachineConfig.st_Q_CameraLightning12.tOutputLocked,
    bProcessedDelayedOutput => gIOFiltered.aCameraLightning[12].bDelayedOutput,
    bProcessedLockedOutput => gIOFiltered.aCameraLightning[12].bLockedOutput); // FB_IO2_OutputCtrl
gIOFiltered.aCameraLightning[12].bStateOutput := aCameraLightControl[12].bProcessedOutput;

// NETWORK 24
bDummyOutput := gIOFiltered.aCameraLightning[12].bLockedOutput;
END_ACTION

ACTION CamerasPower:
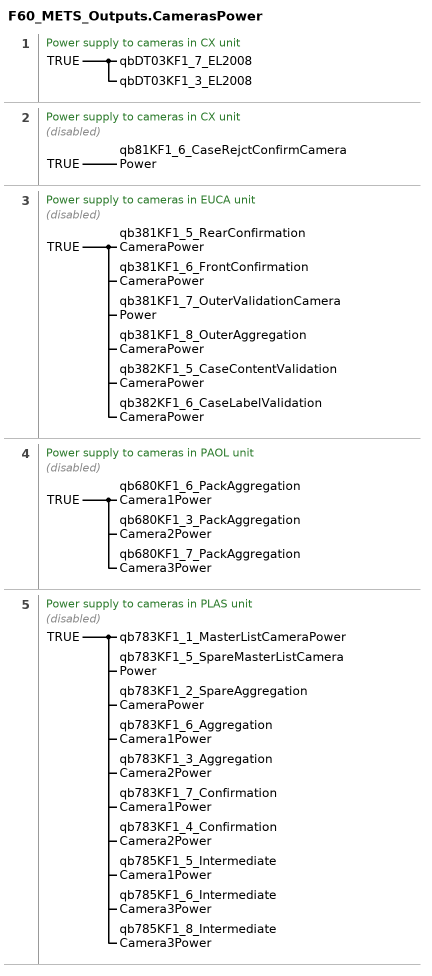
// NETWORK 1
// 					Power supply to cameras in CX unit
//
//
qbDT03KF1_7_EL2008 := TRUE;
qbDT03KF1_3_EL2008 := TRUE;

// NETWORK 2 (disabled)
// 					Power supply to cameras in CX unit
//
//
// qb81KF1_6_CaseRejctConfirmCameraPower := TRUE;

// NETWORK 3 (disabled)
// 					Power supply to cameras in EUCA unit
//
//
// qb381KF1_5_RearConfirmationCameraPower := TRUE;
// qb381KF1_6_FrontConfirmationCameraPower := TRUE;
// qb381KF1_7_OuterValidationCameraPower := TRUE;
// qb381KF1_8_OuterAggregationCameraPower := TRUE;
// qb382KF1_5_CaseContentValidationCameraPower := TRUE;
// qb382KF1_6_CaseLabelValidationCameraPower := TRUE;

// NETWORK 4 (disabled)
// 					Power supply to cameras in PAOL unit
//
//
// qb680KF1_6_PackAggregationCamera1Power := TRUE;
// qb680KF1_3_PackAggregationCamera2Power := TRUE;
// qb680KF1_7_PackAggregationCamera3Power := TRUE;

// NETWORK 5 (disabled)
// 					Power supply to cameras in PLAS unit
//
//
// qb783KF1_1_MasterListCameraPower := TRUE;
// qb783KF1_5_SpareMasterListCameraPower := TRUE;
// qb783KF1_2_SpareAggregationCameraPower := TRUE;
// qb783KF1_6_AggregationCamera1Power := TRUE;
// qb783KF1_3_AggregationCamera2Power := TRUE;
// qb783KF1_7_ConfirmationCamera1Power := TRUE;
// qb783KF1_4_ConfirmationCamera2Power := TRUE;
// qb785KF1_5_IntermediateCamera1Power := TRUE;
// qb785KF1_6_IntermediateCamera3Power := TRUE;
// qb785KF1_8_IntermediateCamera3Power := TRUE;
END_ACTION

ACTION Cylinders:
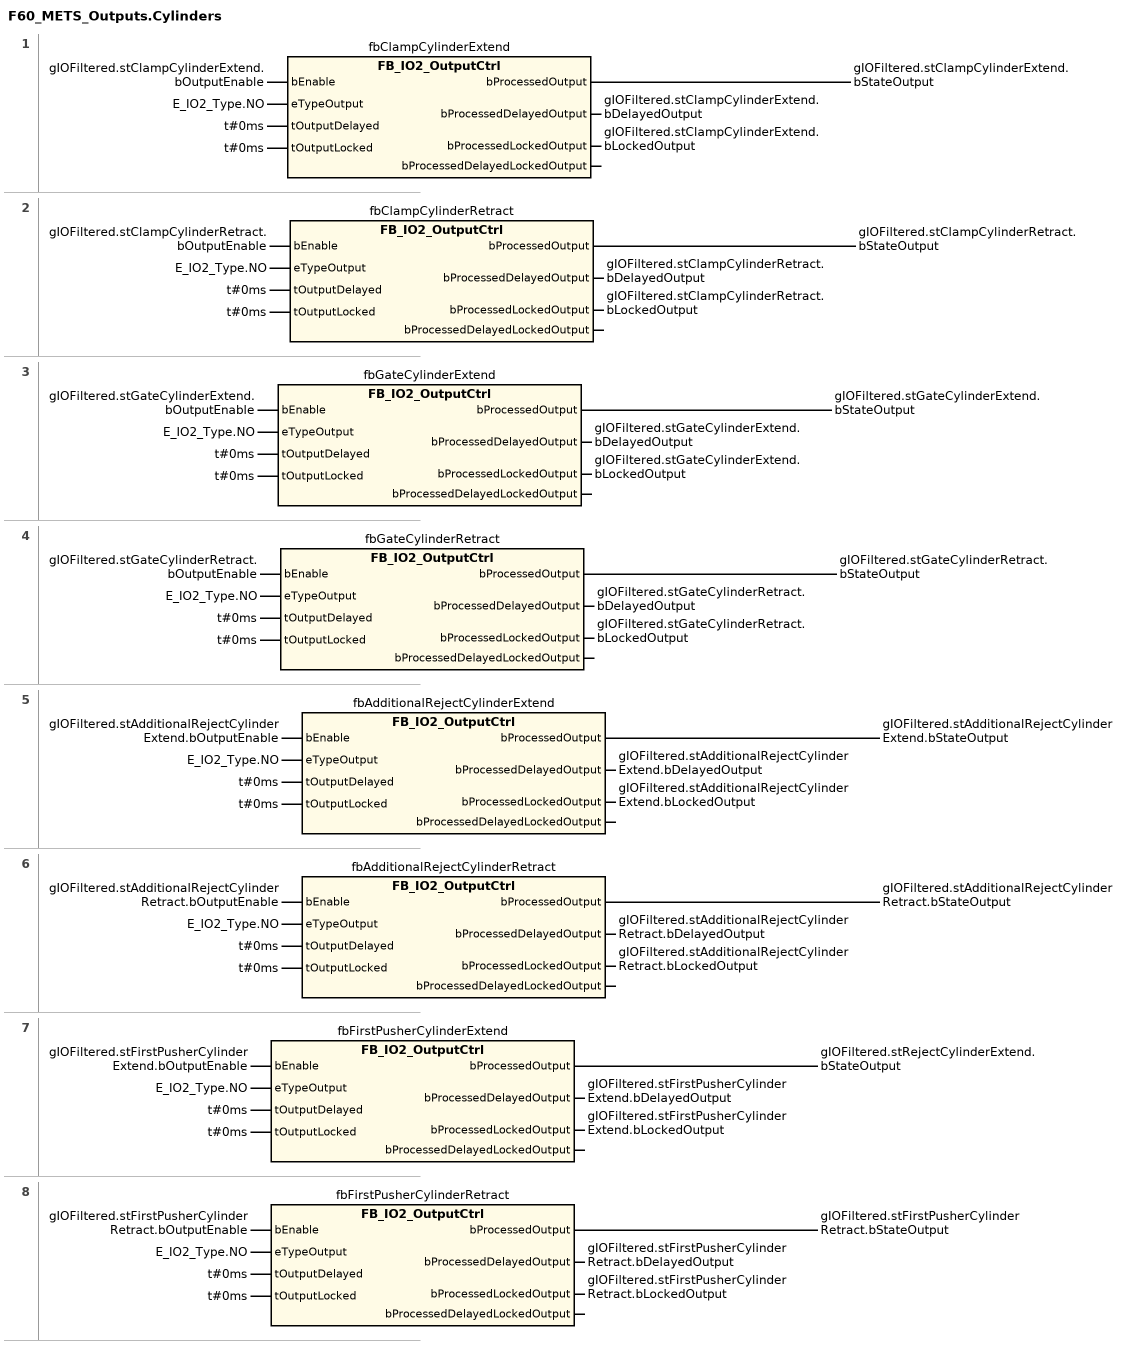
// NETWORK 1
fbClampCylinderExtend(
    bEnable := gIOFiltered.stClampCylinderExtend.bOutputEnable,
    eTypeOutput := E_IO2_Type.NO,
    tOutputDelayed := t#0ms,
    tOutputLocked := t#0ms,
    bProcessedDelayedOutput => gIOFiltered.stClampCylinderExtend.bDelayedOutput,
    bProcessedLockedOutput => gIOFiltered.stClampCylinderExtend.bLockedOutput); // FB_IO2_OutputCtrl
gIOFiltered.stClampCylinderExtend.bStateOutput := fbClampCylinderExtend.bProcessedOutput;

// NETWORK 2
fbClampCylinderRetract(
    bEnable := gIOFiltered.stClampCylinderRetract.bOutputEnable,
    eTypeOutput := E_IO2_Type.NO,
    tOutputDelayed := t#0ms,
    tOutputLocked := t#0ms,
    bProcessedDelayedOutput => gIOFiltered.stClampCylinderRetract.bDelayedOutput,
    bProcessedLockedOutput => gIOFiltered.stClampCylinderRetract.bLockedOutput); // FB_IO2_OutputCtrl
gIOFiltered.stClampCylinderRetract.bStateOutput := fbClampCylinderRetract.bProcessedOutput;

// NETWORK 3
fbGateCylinderExtend(
    bEnable := gIOFiltered.stGateCylinderExtend.bOutputEnable,
    eTypeOutput := E_IO2_Type.NO,
    tOutputDelayed := t#0ms,
    tOutputLocked := t#0ms,
    bProcessedDelayedOutput => gIOFiltered.stGateCylinderExtend.bDelayedOutput,
    bProcessedLockedOutput => gIOFiltered.stGateCylinderExtend.bLockedOutput); // FB_IO2_OutputCtrl
gIOFiltered.stGateCylinderExtend.bStateOutput := fbGateCylinderExtend.bProcessedOutput;

// NETWORK 4
fbGateCylinderRetract(
    bEnable := gIOFiltered.stGateCylinderRetract.bOutputEnable,
    eTypeOutput := E_IO2_Type.NO,
    tOutputDelayed := t#0ms,
    tOutputLocked := t#0ms,
    bProcessedDelayedOutput => gIOFiltered.stGateCylinderRetract.bDelayedOutput,
    bProcessedLockedOutput => gIOFiltered.stGateCylinderRetract.bLockedOutput); // FB_IO2_OutputCtrl
gIOFiltered.stGateCylinderRetract.bStateOutput := fbGateCylinderRetract.bProcessedOutput;

// NETWORK 5
fbAdditionalRejectCylinderExtend(
    bEnable := gIOFiltered.stAdditionalRejectCylinderExtend.bOutputEnable,
    eTypeOutput := E_IO2_Type.NO,
    tOutputDelayed := t#0ms,
    tOutputLocked := t#0ms,
    bProcessedDelayedOutput => gIOFiltered.stAdditionalRejectCylinderExtend.bDelayedOutput,
    bProcessedLockedOutput => gIOFiltered.stAdditionalRejectCylinderExtend.bLockedOutput); // FB_IO2_OutputCtrl
gIOFiltered.stAdditionalRejectCylinderExtend.bStateOutput := fbAdditionalRejectCylinderExtend.bProcessedOutput;

// NETWORK 6
fbAdditionalRejectCylinderRetract(
    bEnable := gIOFiltered.stAdditionalRejectCylinderRetract.bOutputEnable,
    eTypeOutput := E_IO2_Type.NO,
    tOutputDelayed := t#0ms,
    tOutputLocked := t#0ms,
    bProcessedDelayedOutput => gIOFiltered.stAdditionalRejectCylinderRetract.bDelayedOutput,
    bProcessedLockedOutput => gIOFiltered.stAdditionalRejectCylinderRetract.bLockedOutput); // FB_IO2_OutputCtrl
gIOFiltered.stAdditionalRejectCylinderRetract.bStateOutput := fbAdditionalRejectCylinderRetract.bProcessedOutput;

// NETWORK 7
fbFirstPusherCylinderExtend(
    bEnable := gIOFiltered.stFirstPusherCylinderExtend.bOutputEnable,
    eTypeOutput := E_IO2_Type.NO,
    tOutputDelayed := t#0ms,
    tOutputLocked := t#0ms,
    bProcessedDelayedOutput => gIOFiltered.stFirstPusherCylinderExtend.bDelayedOutput,
    bProcessedLockedOutput => gIOFiltered.stFirstPusherCylinderExtend.bLockedOutput); // FB_IO2_OutputCtrl
gIOFiltered.stRejectCylinderExtend.bStateOutput := fbFirstPusherCylinderExtend.bProcessedOutput;

// NETWORK 8
fbFirstPusherCylinderRetract(
    bEnable := gIOFiltered.stFirstPusherCylinderRetract.bOutputEnable,
    eTypeOutput := E_IO2_Type.NO,
    tOutputDelayed := t#0ms,
    tOutputLocked := t#0ms,
    bProcessedDelayedOutput => gIOFiltered.stFirstPusherCylinderRetract.bDelayedOutput,
    bProcessedLockedOutput => gIOFiltered.stFirstPusherCylinderRetract.bLockedOutput); // FB_IO2_OutputCtrl
gIOFiltered.stFirstPusherCylinderRetract.bStateOutput := fbFirstPusherCylinderRetract.bProcessedOutput;

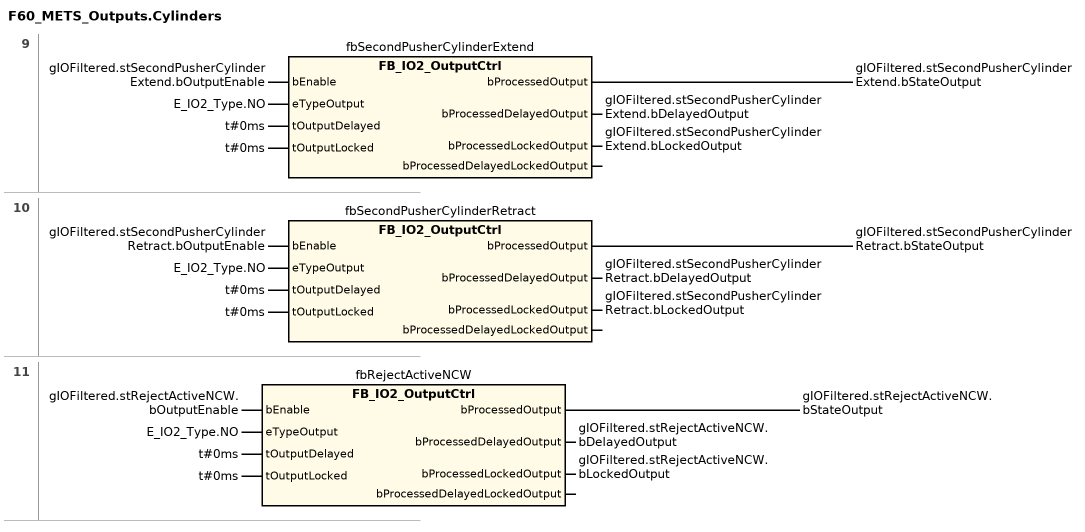
// NETWORK 9
fbSecondPusherCylinderExtend(
    bEnable := gIOFiltered.stSecondPusherCylinderExtend.bOutputEnable,
    eTypeOutput := E_IO2_Type.NO,
    tOutputDelayed := t#0ms,
    tOutputLocked := t#0ms,
    bProcessedDelayedOutput => gIOFiltered.stSecondPusherCylinderExtend.bDelayedOutput,
    bProcessedLockedOutput => gIOFiltered.stSecondPusherCylinderExtend.bLockedOutput); // FB_IO2_OutputCtrl
gIOFiltered.stSecondPusherCylinderExtend.bStateOutput := fbSecondPusherCylinderExtend.bProcessedOutput;

// NETWORK 10
fbSecondPusherCylinderRetract(
    bEnable := gIOFiltered.stSecondPusherCylinderRetract.bOutputEnable,
    eTypeOutput := E_IO2_Type.NO,
    tOutputDelayed := t#0ms,
    tOutputLocked := t#0ms,
    bProcessedDelayedOutput => gIOFiltered.stSecondPusherCylinderRetract.bDelayedOutput,
    bProcessedLockedOutput => gIOFiltered.stSecondPusherCylinderRetract.bLockedOutput); // FB_IO2_OutputCtrl
gIOFiltered.stSecondPusherCylinderRetract.bStateOutput := fbSecondPusherCylinderRetract.bProcessedOutput;

// NETWORK 11
fbRejectActiveNCW(
    bEnable := gIOFiltered.stRejectActiveNCW.bOutputEnable,
    eTypeOutput := E_IO2_Type.NO,
    tOutputDelayed := t#0ms,
    tOutputLocked := t#0ms,
    bProcessedDelayedOutput => gIOFiltered.stRejectActiveNCW.bDelayedOutput,
    bProcessedLockedOutput => gIOFiltered.stRejectActiveNCW.bLockedOutput); // FB_IO2_OutputCtrl
gIOFiltered.stRejectActiveNCW.bStateOutput := fbRejectActiveNCW.bProcessedOutput;
END_ACTION

ACTION Drives:
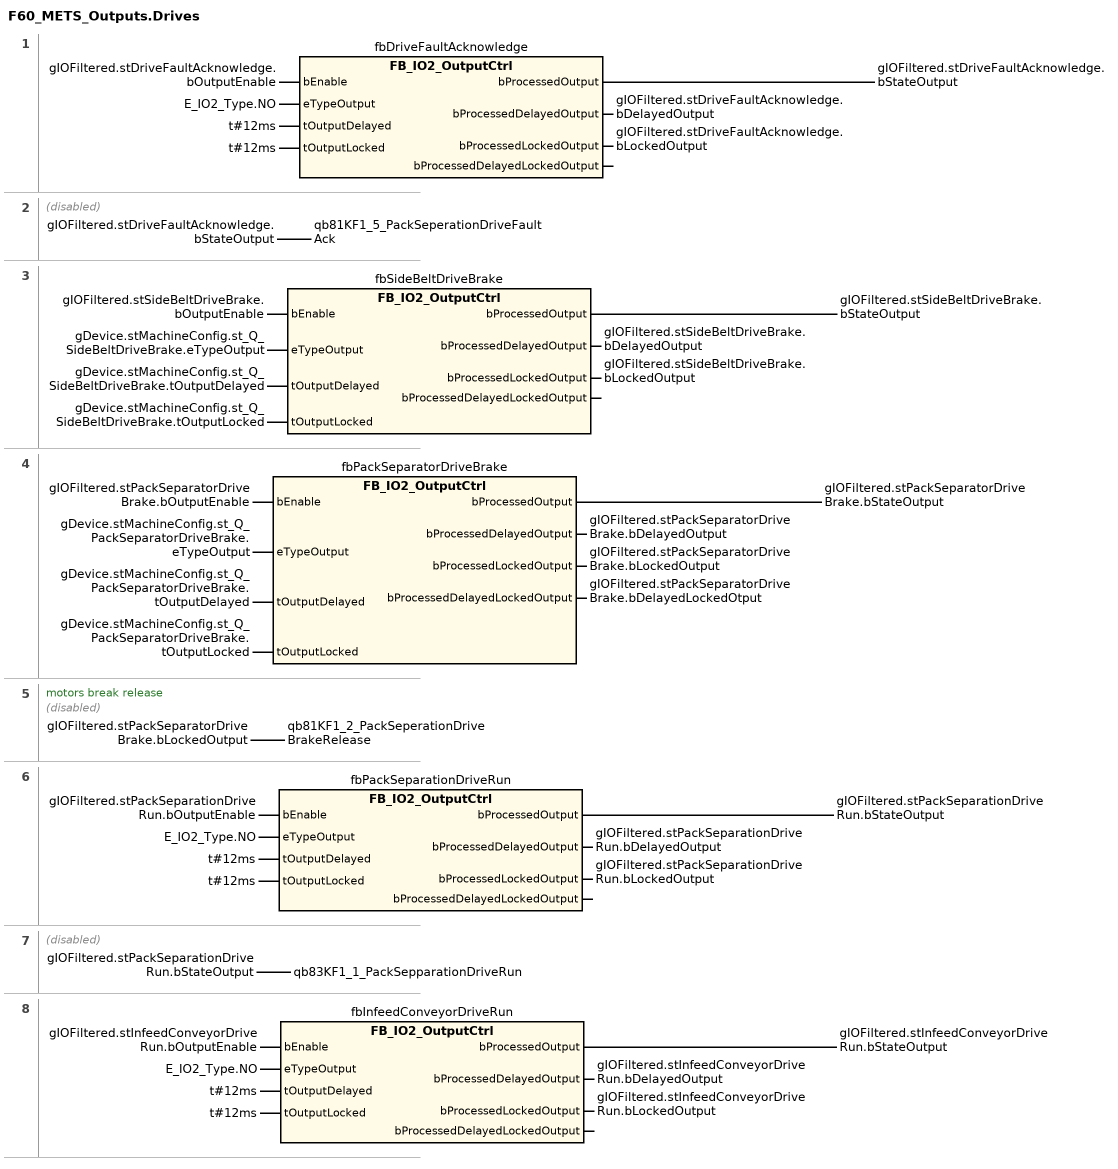
// NETWORK 1
fbDriveFaultAcknowledge(
    bEnable := gIOFiltered.stDriveFaultAcknowledge.bOutputEnable,
    eTypeOutput := E_IO2_Type.NO,
    tOutputDelayed := t#12ms,
    tOutputLocked := t#12ms,
    bProcessedDelayedOutput => gIOFiltered.stDriveFaultAcknowledge.bDelayedOutput,
    bProcessedLockedOutput => gIOFiltered.stDriveFaultAcknowledge.bLockedOutput); // FB_IO2_OutputCtrl
gIOFiltered.stDriveFaultAcknowledge.bStateOutput := fbDriveFaultAcknowledge.bProcessedOutput;

// NETWORK 2 (disabled)
// qb81KF1_5_PackSeperationDriveFaultAck := gIOFiltered.stDriveFaultAcknowledge.bStateOutput;

// NETWORK 3
fbSideBeltDriveBrake(
    bEnable := gIOFiltered.stSideBeltDriveBrake.bOutputEnable,
    eTypeOutput := gDevice.stMachineConfig.st_Q_SideBeltDriveBrake.eTypeOutput,
    tOutputDelayed := gDevice.stMachineConfig.st_Q_SideBeltDriveBrake.tOutputDelayed,
    tOutputLocked := gDevice.stMachineConfig.st_Q_SideBeltDriveBrake.tOutputLocked,
    bProcessedDelayedOutput => gIOFiltered.stSideBeltDriveBrake.bDelayedOutput,
    bProcessedLockedOutput => gIOFiltered.stSideBeltDriveBrake.bLockedOutput); // FB_IO2_OutputCtrl
gIOFiltered.stSideBeltDriveBrake.bStateOutput := fbSideBeltDriveBrake.bProcessedOutput;

// NETWORK 4
fbPackSeparatorDriveBrake(
    bEnable := gIOFiltered.stPackSeparatorDriveBrake.bOutputEnable,
    eTypeOutput := gDevice.stMachineConfig.st_Q_PackSeparatorDriveBrake.eTypeOutput,
    tOutputDelayed := gDevice.stMachineConfig.st_Q_PackSeparatorDriveBrake.tOutputDelayed,
    tOutputLocked := gDevice.stMachineConfig.st_Q_PackSeparatorDriveBrake.tOutputLocked,
    bProcessedDelayedOutput => gIOFiltered.stPackSeparatorDriveBrake.bDelayedOutput,
    bProcessedLockedOutput => gIOFiltered.stPackSeparatorDriveBrake.bLockedOutput,
    bProcessedDelayedLockedOutput => gIOFiltered.stPackSeparatorDriveBrake.bDelayedLockedOtput); // FB_IO2_OutputCtrl
gIOFiltered.stPackSeparatorDriveBrake.bStateOutput := fbPackSeparatorDriveBrake.bProcessedOutput;

// NETWORK 5 (disabled)
// motors break release
// qb81KF1_2_PackSeperationDriveBrakeRelease := gIOFiltered.stPackSeparatorDriveBrake.bLockedOutput;

// NETWORK 6
fbPackSeparationDriveRun(
    bEnable := gIOFiltered.stPackSeparationDriveRun.bOutputEnable,
    eTypeOutput := E_IO2_Type.NO,
    tOutputDelayed := t#12ms,
    tOutputLocked := t#12ms,
    bProcessedDelayedOutput => gIOFiltered.stPackSeparationDriveRun.bDelayedOutput,
    bProcessedLockedOutput => gIOFiltered.stPackSeparationDriveRun.bLockedOutput); // FB_IO2_OutputCtrl
gIOFiltered.stPackSeparationDriveRun.bStateOutput := fbPackSeparationDriveRun.bProcessedOutput;

// NETWORK 7 (disabled)
// qb83KF1_1_PackSepparationDriveRun := gIOFiltered.stPackSeparationDriveRun.bStateOutput;

// NETWORK 8
fbInfeedConveyorDriveRun(
    bEnable := gIOFiltered.stInfeedConveyorDriveRun.bOutputEnable,
    eTypeOutput := E_IO2_Type.NO,
    tOutputDelayed := t#12ms,
    tOutputLocked := t#12ms,
    bProcessedDelayedOutput => gIOFiltered.stInfeedConveyorDriveRun.bDelayedOutput,
    bProcessedLockedOutput => gIOFiltered.stInfeedConveyorDriveRun.bLockedOutput); // FB_IO2_OutputCtrl
gIOFiltered.stInfeedConveyorDriveRun.bStateOutput := fbInfeedConveyorDriveRun.bProcessedOutput;
END_ACTION

ACTION Labellers:
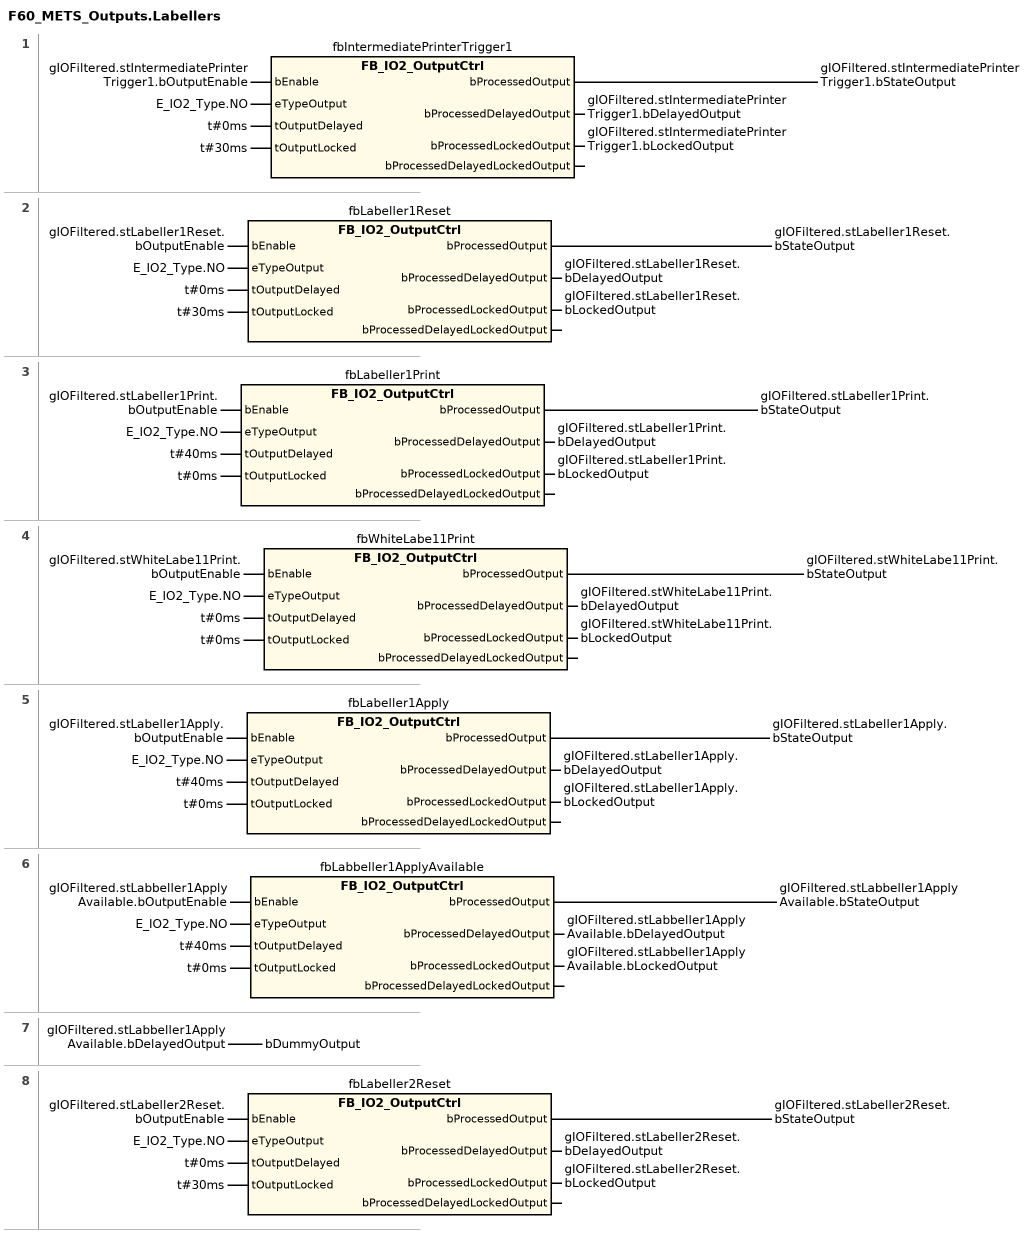
// NETWORK 1
fbIntermediatePrinterTrigger1(
    bEnable := gIOFiltered.stIntermediatePrinterTrigger1.bOutputEnable,
    eTypeOutput := E_IO2_Type.NO,
    tOutputDelayed := t#0ms,
    tOutputLocked := t#30ms,
    bProcessedDelayedOutput => gIOFiltered.stIntermediatePrinterTrigger1.bDelayedOutput,
    bProcessedLockedOutput => gIOFiltered.stIntermediatePrinterTrigger1.bLockedOutput); // FB_IO2_OutputCtrl
gIOFiltered.stIntermediatePrinterTrigger1.bStateOutput := fbIntermediatePrinterTrigger1.bProcessedOutput;

// NETWORK 2
fbLabeller1Reset(
    bEnable := gIOFiltered.stLabeller1Reset.bOutputEnable,
    eTypeOutput := E_IO2_Type.NO,
    tOutputDelayed := t#0ms,
    tOutputLocked := t#30ms,
    bProcessedDelayedOutput => gIOFiltered.stLabeller1Reset.bDelayedOutput,
    bProcessedLockedOutput => gIOFiltered.stLabeller1Reset.bLockedOutput); // FB_IO2_OutputCtrl
gIOFiltered.stLabeller1Reset.bStateOutput := fbLabeller1Reset.bProcessedOutput;

// NETWORK 3
fbLabeller1Print(
    bEnable := gIOFiltered.stLabeller1Print.bOutputEnable,
    eTypeOutput := E_IO2_Type.NO,
    tOutputDelayed := t#40ms,
    tOutputLocked := t#0ms,
    bProcessedDelayedOutput => gIOFiltered.stLabeller1Print.bDelayedOutput,
    bProcessedLockedOutput => gIOFiltered.stLabeller1Print.bLockedOutput); // FB_IO2_OutputCtrl
gIOFiltered.stLabeller1Print.bStateOutput := fbLabeller1Print.bProcessedOutput;

// NETWORK 4
fbWhiteLabe11Print(
    bEnable := gIOFiltered.stWhiteLabe11Print.bOutputEnable,
    eTypeOutput := E_IO2_Type.NO,
    tOutputDelayed := t#0ms,
    tOutputLocked := t#0ms,
    bProcessedDelayedOutput => gIOFiltered.stWhiteLabe11Print.bDelayedOutput,
    bProcessedLockedOutput => gIOFiltered.stWhiteLabe11Print.bLockedOutput); // FB_IO2_OutputCtrl
gIOFiltered.stWhiteLabe11Print.bStateOutput := fbWhiteLabe11Print.bProcessedOutput;

// NETWORK 5
fbLabeller1Apply(
    bEnable := gIOFiltered.stLabeller1Apply.bOutputEnable,
    eTypeOutput := E_IO2_Type.NO,
    tOutputDelayed := t#40ms,
    tOutputLocked := t#0ms,
    bProcessedDelayedOutput => gIOFiltered.stLabeller1Apply.bDelayedOutput,
    bProcessedLockedOutput => gIOFiltered.stLabeller1Apply.bLockedOutput); // FB_IO2_OutputCtrl
gIOFiltered.stLabeller1Apply.bStateOutput := fbLabeller1Apply.bProcessedOutput;

// NETWORK 6
fbLabbeller1ApplyAvailable(
    bEnable := gIOFiltered.stLabbeller1ApplyAvailable.bOutputEnable,
    eTypeOutput := E_IO2_Type.NO,
    tOutputDelayed := t#40ms,
    tOutputLocked := t#0ms,
    bProcessedDelayedOutput => gIOFiltered.stLabbeller1ApplyAvailable.bDelayedOutput,
    bProcessedLockedOutput => gIOFiltered.stLabbeller1ApplyAvailable.bLockedOutput); // FB_IO2_OutputCtrl
gIOFiltered.stLabbeller1ApplyAvailable.bStateOutput := fbLabbeller1ApplyAvailable.bProcessedOutput;

// NETWORK 7
bDummyOutput := gIOFiltered.stLabbeller1ApplyAvailable.bDelayedOutput;

// NETWORK 8
fbLabeller2Reset(
    bEnable := gIOFiltered.stLabeller2Reset.bOutputEnable,
    eTypeOutput := E_IO2_Type.NO,
    tOutputDelayed := t#0ms,
    tOutputLocked := t#30ms,
    bProcessedDelayedOutput => gIOFiltered.stLabeller2Reset.bDelayedOutput,
    bProcessedLockedOutput => gIOFiltered.stLabeller2Reset.bLockedOutput); // FB_IO2_OutputCtrl
gIOFiltered.stLabeller2Reset.bStateOutput := fbLabeller2Reset.bProcessedOutput;

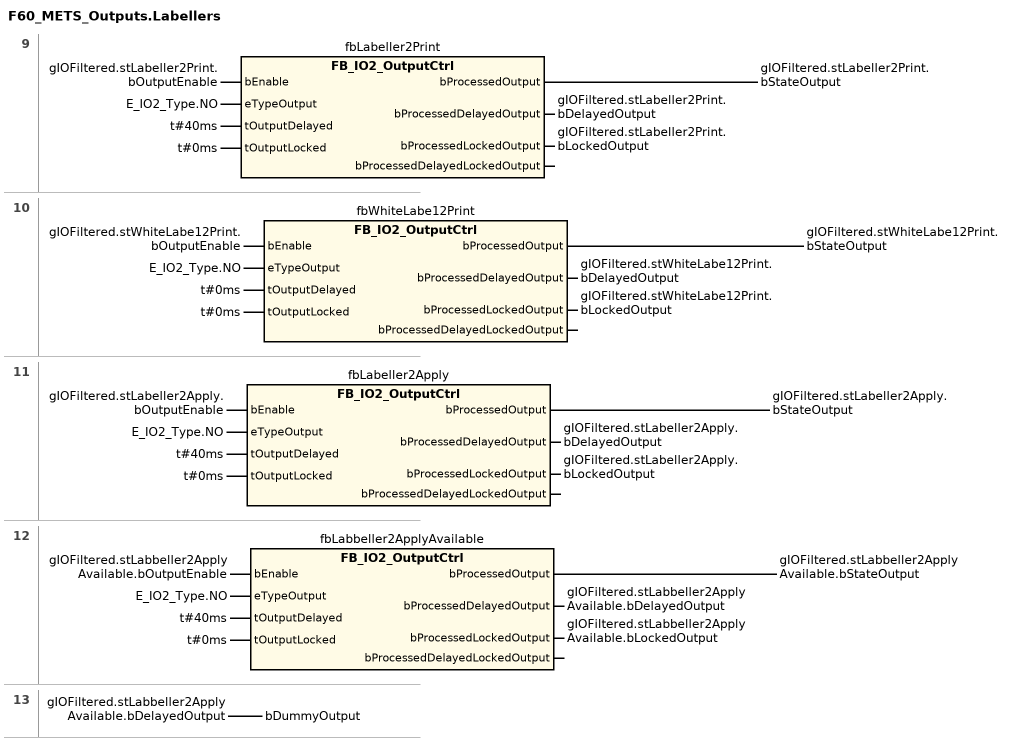
// NETWORK 9
fbLabeller2Print(
    bEnable := gIOFiltered.stLabeller2Print.bOutputEnable,
    eTypeOutput := E_IO2_Type.NO,
    tOutputDelayed := t#40ms,
    tOutputLocked := t#0ms,
    bProcessedDelayedOutput => gIOFiltered.stLabeller2Print.bDelayedOutput,
    bProcessedLockedOutput => gIOFiltered.stLabeller2Print.bLockedOutput); // FB_IO2_OutputCtrl
gIOFiltered.stLabeller2Print.bStateOutput := fbLabeller2Print.bProcessedOutput;

// NETWORK 10
fbWhiteLabe12Print(
    bEnable := gIOFiltered.stWhiteLabe12Print.bOutputEnable,
    eTypeOutput := E_IO2_Type.NO,
    tOutputDelayed := t#0ms,
    tOutputLocked := t#0ms,
    bProcessedDelayedOutput => gIOFiltered.stWhiteLabe12Print.bDelayedOutput,
    bProcessedLockedOutput => gIOFiltered.stWhiteLabe12Print.bLockedOutput); // FB_IO2_OutputCtrl
gIOFiltered.stWhiteLabe12Print.bStateOutput := fbWhiteLabe12Print.bProcessedOutput;

// NETWORK 11
fbLabeller2Apply(
    bEnable := gIOFiltered.stLabeller2Apply.bOutputEnable,
    eTypeOutput := E_IO2_Type.NO,
    tOutputDelayed := t#40ms,
    tOutputLocked := t#0ms,
    bProcessedDelayedOutput => gIOFiltered.stLabeller2Apply.bDelayedOutput,
    bProcessedLockedOutput => gIOFiltered.stLabeller2Apply.bLockedOutput); // FB_IO2_OutputCtrl
gIOFiltered.stLabeller2Apply.bStateOutput := fbLabeller2Apply.bProcessedOutput;

// NETWORK 12
fbLabbeller2ApplyAvailable(
    bEnable := gIOFiltered.stLabbeller2ApplyAvailable.bOutputEnable,
    eTypeOutput := E_IO2_Type.NO,
    tOutputDelayed := t#40ms,
    tOutputLocked := t#0ms,
    bProcessedDelayedOutput => gIOFiltered.stLabbeller2ApplyAvailable.bDelayedOutput,
    bProcessedLockedOutput => gIOFiltered.stLabbeller2ApplyAvailable.bLockedOutput); // FB_IO2_OutputCtrl
gIOFiltered.stLabbeller2ApplyAvailable.bStateOutput := fbLabbeller2ApplyAvailable.bProcessedOutput;

// NETWORK 13
bDummyOutput := gIOFiltered.stLabbeller2ApplyAvailable.bDelayedOutput;
END_ACTION

ACTION LightPole:
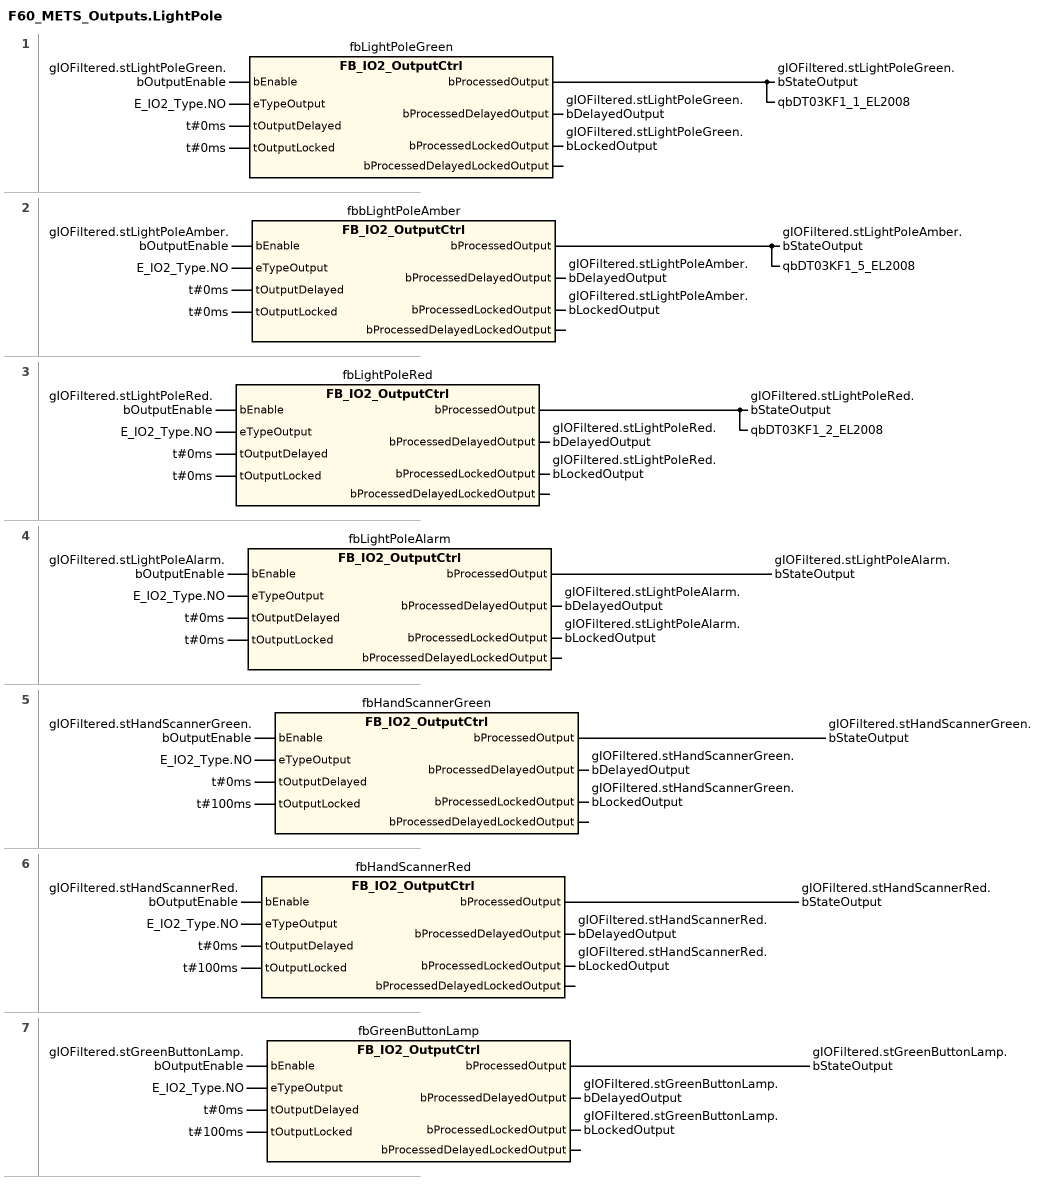
// NETWORK 1
fbLightPoleGreen(
    bEnable := gIOFiltered.stLightPoleGreen.bOutputEnable,
    eTypeOutput := E_IO2_Type.NO,
    tOutputDelayed := t#0ms,
    tOutputLocked := t#0ms,
    bProcessedDelayedOutput => gIOFiltered.stLightPoleGreen.bDelayedOutput,
    bProcessedLockedOutput => gIOFiltered.stLightPoleGreen.bLockedOutput); // FB_IO2_OutputCtrl
gIOFiltered.stLightPoleGreen.bStateOutput := fbLightPoleGreen.bProcessedOutput;
qbDT03KF1_1_EL2008 := fbLightPoleGreen.bProcessedOutput;

// NETWORK 2
fbbLightPoleAmber(
    bEnable := gIOFiltered.stLightPoleAmber.bOutputEnable,
    eTypeOutput := E_IO2_Type.NO,
    tOutputDelayed := t#0ms,
    tOutputLocked := t#0ms,
    bProcessedDelayedOutput => gIOFiltered.stLightPoleAmber.bDelayedOutput,
    bProcessedLockedOutput => gIOFiltered.stLightPoleAmber.bLockedOutput); // FB_IO2_OutputCtrl
gIOFiltered.stLightPoleAmber.bStateOutput := fbbLightPoleAmber.bProcessedOutput;
qbDT03KF1_5_EL2008 := fbbLightPoleAmber.bProcessedOutput;

// NETWORK 3
fbLightPoleRed(
    bEnable := gIOFiltered.stLightPoleRed.bOutputEnable,
    eTypeOutput := E_IO2_Type.NO,
    tOutputDelayed := t#0ms,
    tOutputLocked := t#0ms,
    bProcessedDelayedOutput => gIOFiltered.stLightPoleRed.bDelayedOutput,
    bProcessedLockedOutput => gIOFiltered.stLightPoleRed.bLockedOutput); // FB_IO2_OutputCtrl
gIOFiltered.stLightPoleRed.bStateOutput := fbLightPoleRed.bProcessedOutput;
qbDT03KF1_2_EL2008 := fbLightPoleRed.bProcessedOutput;

// NETWORK 4
fbLightPoleAlarm(
    bEnable := gIOFiltered.stLightPoleAlarm.bOutputEnable,
    eTypeOutput := E_IO2_Type.NO,
    tOutputDelayed := t#0ms,
    tOutputLocked := t#0ms,
    bProcessedDelayedOutput => gIOFiltered.stLightPoleAlarm.bDelayedOutput,
    bProcessedLockedOutput => gIOFiltered.stLightPoleAlarm.bLockedOutput); // FB_IO2_OutputCtrl
gIOFiltered.stLightPoleAlarm.bStateOutput := fbLightPoleAlarm.bProcessedOutput;

// NETWORK 5
fbHandScannerGreen(
    bEnable := gIOFiltered.stHandScannerGreen.bOutputEnable,
    eTypeOutput := E_IO2_Type.NO,
    tOutputDelayed := t#0ms,
    tOutputLocked := t#100ms,
    bProcessedDelayedOutput => gIOFiltered.stHandScannerGreen.bDelayedOutput,
    bProcessedLockedOutput => gIOFiltered.stHandScannerGreen.bLockedOutput); // FB_IO2_OutputCtrl
gIOFiltered.stHandScannerGreen.bStateOutput := fbHandScannerGreen.bProcessedOutput;

// NETWORK 6
fbHandScannerRed(
    bEnable := gIOFiltered.stHandScannerRed.bOutputEnable,
    eTypeOutput := E_IO2_Type.NO,
    tOutputDelayed := t#0ms,
    tOutputLocked := t#100ms,
    bProcessedDelayedOutput => gIOFiltered.stHandScannerRed.bDelayedOutput,
    bProcessedLockedOutput => gIOFiltered.stHandScannerRed.bLockedOutput); // FB_IO2_OutputCtrl
gIOFiltered.stHandScannerRed.bStateOutput := fbHandScannerRed.bProcessedOutput;

// NETWORK 7
fbGreenButtonLamp(
    bEnable := gIOFiltered.stGreenButtonLamp.bOutputEnable,
    eTypeOutput := E_IO2_Type.NO,
    tOutputDelayed := t#0ms,
    tOutputLocked := t#100ms,
    bProcessedDelayedOutput => gIOFiltered.stGreenButtonLamp.bDelayedOutput,
    bProcessedLockedOutput => gIOFiltered.stGreenButtonLamp.bLockedOutput); // FB_IO2_OutputCtrl
gIOFiltered.stGreenButtonLamp.bStateOutput := fbGreenButtonLamp.bProcessedOutput;
END_ACTION

ACTION Safety:
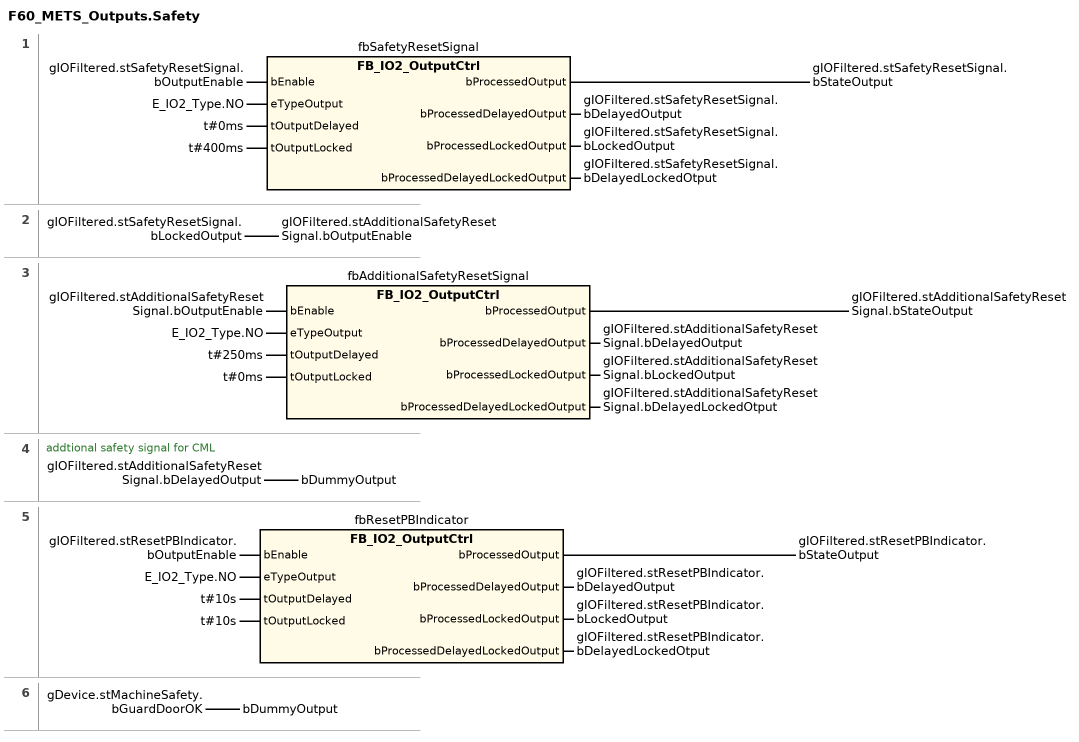
// NETWORK 1
fbSafetyResetSignal(
    bEnable := gIOFiltered.stSafetyResetSignal.bOutputEnable,
    eTypeOutput := E_IO2_Type.NO,
    tOutputDelayed := t#0ms,
    tOutputLocked := t#400ms,
    bProcessedDelayedOutput => gIOFiltered.stSafetyResetSignal.bDelayedOutput,
    bProcessedLockedOutput => gIOFiltered.stSafetyResetSignal.bLockedOutput,
    bProcessedDelayedLockedOutput => gIOFiltered.stSafetyResetSignal.bDelayedLockedOtput); // FB_IO2_OutputCtrl
gIOFiltered.stSafetyResetSignal.bStateOutput := fbSafetyResetSignal.bProcessedOutput;

// NETWORK 2
gIOFiltered.stAdditionalSafetyResetSignal.bOutputEnable := gIOFiltered.stSafetyResetSignal.bLockedOutput;

// NETWORK 3
fbAdditionalSafetyResetSignal(
    bEnable := gIOFiltered.stAdditionalSafetyResetSignal.bOutputEnable,
    eTypeOutput := E_IO2_Type.NO,
    tOutputDelayed := t#250ms,
    tOutputLocked := t#0ms,
    bProcessedDelayedOutput => gIOFiltered.stAdditionalSafetyResetSignal.bDelayedOutput,
    bProcessedLockedOutput => gIOFiltered.stAdditionalSafetyResetSignal.bLockedOutput,
    bProcessedDelayedLockedOutput => gIOFiltered.stAdditionalSafetyResetSignal.bDelayedLockedOtput); // FB_IO2_OutputCtrl
gIOFiltered.stAdditionalSafetyResetSignal.bStateOutput := fbAdditionalSafetyResetSignal.bProcessedOutput;

// NETWORK 4
// addtional safety signal for CML
bDummyOutput := gIOFiltered.stAdditionalSafetyResetSignal.bDelayedOutput;

// NETWORK 5
fbResetPBIndicator(
    bEnable := gIOFiltered.stResetPBIndicator.bOutputEnable,
    eTypeOutput := E_IO2_Type.NO,
    tOutputDelayed := t#10s,
    tOutputLocked := t#10s,
    bProcessedDelayedOutput => gIOFiltered.stResetPBIndicator.bDelayedOutput,
    bProcessedLockedOutput => gIOFiltered.stResetPBIndicator.bLockedOutput,
    bProcessedDelayedLockedOutput => gIOFiltered.stResetPBIndicator.bDelayedLockedOtput); // FB_IO2_OutputCtrl
gIOFiltered.stResetPBIndicator.bStateOutput := fbResetPBIndicator.bProcessedOutput;

// NETWORK 6
bDummyOutput := gDevice.stMachineSafety.bGuardDoorOK;
END_ACTION

ACTION SystemRun:
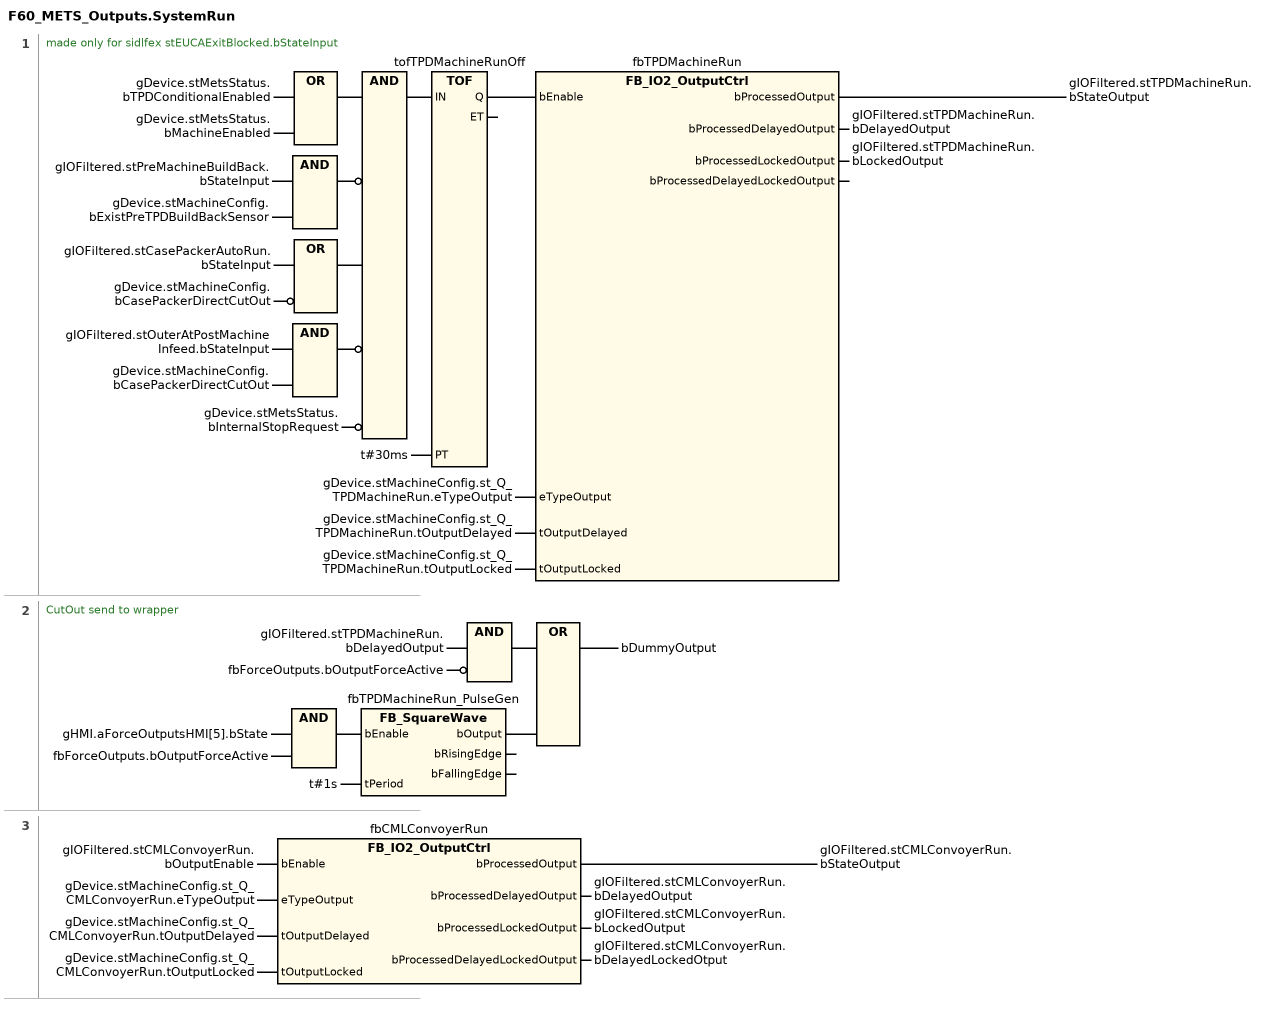
// NETWORK 1
// made only for sidlfex stEUCAExitBlocked.bStateInput
tofTPDMachineRunOff(IN := (gDevice.stMetsStatus.bTPDConditionalEnabled OR gDevice.stMetsStatus.bMachineEnabled) AND NOT (gIOFiltered.stPreMachineBuildBack.bStateInput AND gDevice.stMachineConfig.bExistPreTPDBuildBackSensor) AND (gIOFiltered.stCasePackerAutoRun.bStateInput OR NOT gDevice.stMachineConfig.bCasePackerDirectCutOut) AND NOT (gIOFiltered.stOuterAtPostMachineInfeed.bStateInput AND gDevice.stMachineConfig.bCasePackerDirectCutOut) AND NOT gDevice.stMetsStatus.bInternalStopRequest, PT := t#30ms); // TOF
fbTPDMachineRun(
    bEnable := tofTPDMachineRunOff.Q,
    eTypeOutput := gDevice.stMachineConfig.st_Q_TPDMachineRun.eTypeOutput,
    tOutputDelayed := gDevice.stMachineConfig.st_Q_TPDMachineRun.tOutputDelayed,
    tOutputLocked := gDevice.stMachineConfig.st_Q_TPDMachineRun.tOutputLocked,
    bProcessedDelayedOutput => gIOFiltered.stTPDMachineRun.bDelayedOutput,
    bProcessedLockedOutput => gIOFiltered.stTPDMachineRun.bLockedOutput); // FB_IO2_OutputCtrl
gIOFiltered.stTPDMachineRun.bStateOutput := fbTPDMachineRun.bProcessedOutput;

// NETWORK 2
// CutOut send to wrapper
fbTPDMachineRun_PulseGen(bEnable := gHMI.aForceOutputsHMI[5].bState AND fbForceOutputs.bOutputForceActive, tPeriod := t#1s); // FB_SquareWave
bDummyOutput := gIOFiltered.stTPDMachineRun.bDelayedOutput AND NOT fbForceOutputs.bOutputForceActive OR fbTPDMachineRun_PulseGen.bOutput;

// NETWORK 3
fbCMLConvoyerRun(
    bEnable := gIOFiltered.stCMLConvoyerRun.bOutputEnable,
    eTypeOutput := gDevice.stMachineConfig.st_Q_CMLConvoyerRun.eTypeOutput,
    tOutputDelayed := gDevice.stMachineConfig.st_Q_CMLConvoyerRun.tOutputDelayed,
    tOutputLocked := gDevice.stMachineConfig.st_Q_CMLConvoyerRun.tOutputLocked,
    bProcessedDelayedOutput => gIOFiltered.stCMLConvoyerRun.bDelayedOutput,
    bProcessedLockedOutput => gIOFiltered.stCMLConvoyerRun.bLockedOutput,
    bProcessedDelayedLockedOutput => gIOFiltered.stCMLConvoyerRun.bDelayedLockedOtput); // FB_IO2_OutputCtrl
gIOFiltered.stCMLConvoyerRun.bStateOutput := fbCMLConvoyerRun.bProcessedOutput;

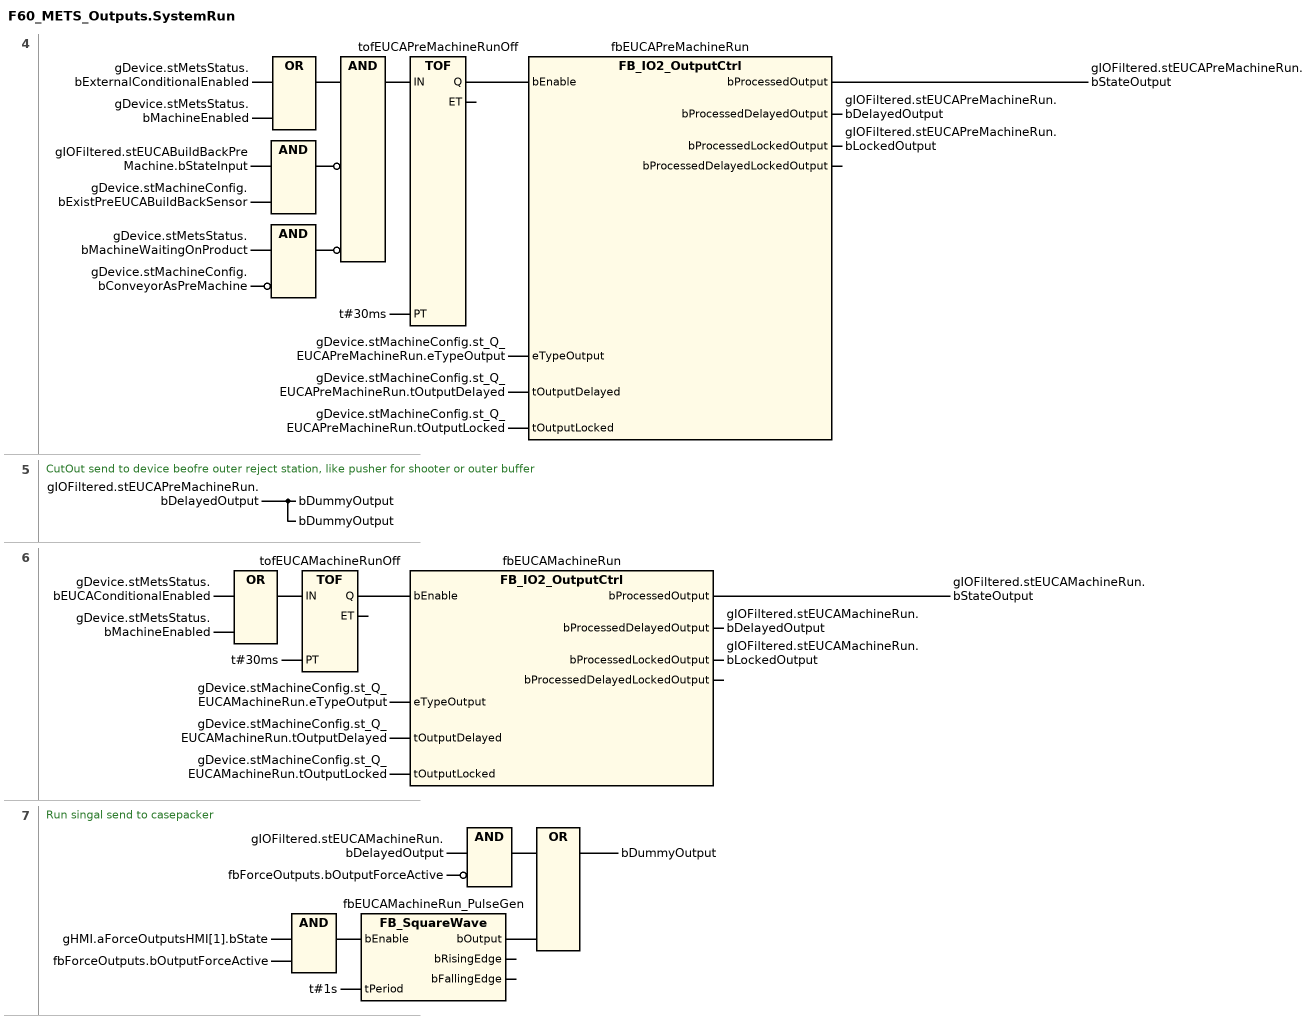
// NETWORK 4
tofEUCAPreMachineRunOff(IN := (gDevice.stMetsStatus.bExternalConditionalEnabled OR gDevice.stMetsStatus.bMachineEnabled) AND NOT (gIOFiltered.stEUCABuildBackPreMachine.bStateInput AND gDevice.stMachineConfig.bExistPreEUCABuildBackSensor) AND NOT (gDevice.stMetsStatus.bMachineWaitingOnProduct AND NOT gDevice.stMachineConfig.bConveyorAsPreMachine), PT := t#30ms); // TOF
fbEUCAPreMachineRun(
    bEnable := tofEUCAPreMachineRunOff.Q,
    eTypeOutput := gDevice.stMachineConfig.st_Q_EUCAPreMachineRun.eTypeOutput,
    tOutputDelayed := gDevice.stMachineConfig.st_Q_EUCAPreMachineRun.tOutputDelayed,
    tOutputLocked := gDevice.stMachineConfig.st_Q_EUCAPreMachineRun.tOutputLocked,
    bProcessedDelayedOutput => gIOFiltered.stEUCAPreMachineRun.bDelayedOutput,
    bProcessedLockedOutput => gIOFiltered.stEUCAPreMachineRun.bLockedOutput); // FB_IO2_OutputCtrl
gIOFiltered.stEUCAPreMachineRun.bStateOutput := fbEUCAPreMachineRun.bProcessedOutput;

// NETWORK 5
// CutOut send to device beofre outer reject station, like pusher for shooter or outer buffer
bDummyOutput := gIOFiltered.stEUCAPreMachineRun.bDelayedOutput;
bDummyOutput := gIOFiltered.stEUCAPreMachineRun.bDelayedOutput;

// NETWORK 6
tofEUCAMachineRunOff(IN := gDevice.stMetsStatus.bEUCAConditionalEnabled OR gDevice.stMetsStatus.bMachineEnabled, PT := t#30ms); // TOF
fbEUCAMachineRun(
    bEnable := tofEUCAMachineRunOff.Q,
    eTypeOutput := gDevice.stMachineConfig.st_Q_EUCAMachineRun.eTypeOutput,
    tOutputDelayed := gDevice.stMachineConfig.st_Q_EUCAMachineRun.tOutputDelayed,
    tOutputLocked := gDevice.stMachineConfig.st_Q_EUCAMachineRun.tOutputLocked,
    bProcessedDelayedOutput => gIOFiltered.stEUCAMachineRun.bDelayedOutput,
    bProcessedLockedOutput => gIOFiltered.stEUCAMachineRun.bLockedOutput); // FB_IO2_OutputCtrl
gIOFiltered.stEUCAMachineRun.bStateOutput := fbEUCAMachineRun.bProcessedOutput;

// NETWORK 7
// Run singal send to casepacker
fbEUCAMachineRun_PulseGen(bEnable := gHMI.aForceOutputsHMI[1].bState AND fbForceOutputs.bOutputForceActive, tPeriod := t#1s); // FB_SquareWave
bDummyOutput := gIOFiltered.stEUCAMachineRun.bDelayedOutput AND NOT fbForceOutputs.bOutputForceActive OR fbEUCAMachineRun_PulseGen.bOutput;
END_ACTION

ACTION Validation:
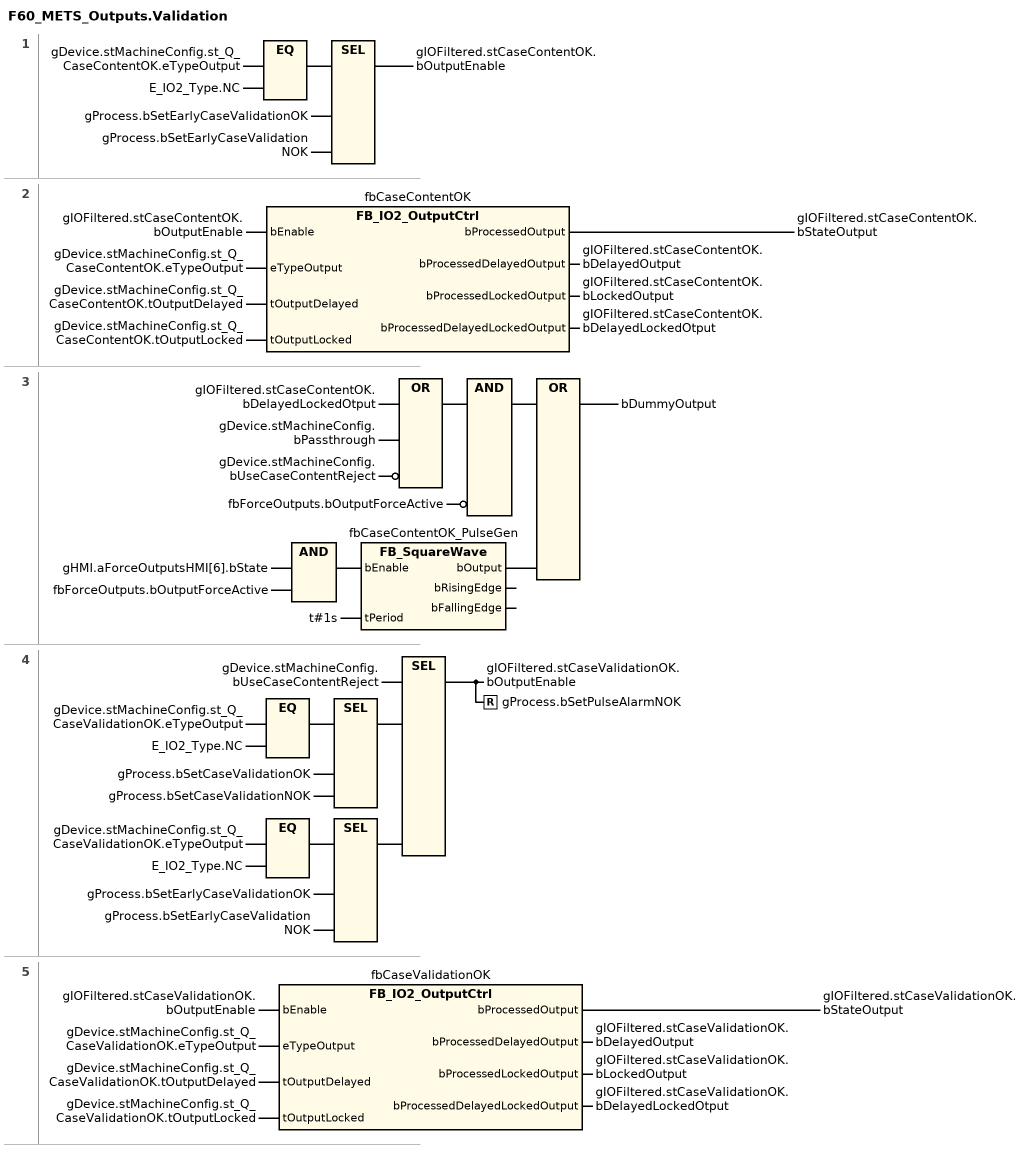
// NETWORK 1
gIOFiltered.stCaseContentOK.bOutputEnable := SEL(gDevice.stMachineConfig.st_Q_CaseContentOK.eTypeOutput = E_IO2_Type.NC, gProcess.bSetEarlyCaseValidationOK, gProcess.bSetEarlyCaseValidationNOK);

// NETWORK 2
fbCaseContentOK(
    bEnable := gIOFiltered.stCaseContentOK.bOutputEnable,
    eTypeOutput := gDevice.stMachineConfig.st_Q_CaseContentOK.eTypeOutput,
    tOutputDelayed := gDevice.stMachineConfig.st_Q_CaseContentOK.tOutputDelayed,
    tOutputLocked := gDevice.stMachineConfig.st_Q_CaseContentOK.tOutputLocked,
    bProcessedDelayedOutput => gIOFiltered.stCaseContentOK.bDelayedOutput,
    bProcessedLockedOutput => gIOFiltered.stCaseContentOK.bLockedOutput,
    bProcessedDelayedLockedOutput => gIOFiltered.stCaseContentOK.bDelayedLockedOtput); // FB_IO2_OutputCtrl
gIOFiltered.stCaseContentOK.bStateOutput := fbCaseContentOK.bProcessedOutput;

// NETWORK 3
fbCaseContentOK_PulseGen(bEnable := gHMI.aForceOutputsHMI[6].bState AND fbForceOutputs.bOutputForceActive, tPeriod := t#1s); // FB_SquareWave
bDummyOutput := (gIOFiltered.stCaseContentOK.bDelayedLockedOtput OR gDevice.stMachineConfig.bPassthrough OR NOT gDevice.stMachineConfig.bUseCaseContentReject) AND NOT fbForceOutputs.bOutputForceActive OR fbCaseContentOK_PulseGen.bOutput;

// NETWORK 4
_w1 := SEL(gDevice.stMachineConfig.bUseCaseContentReject, SEL(gDevice.stMachineConfig.st_Q_CaseValidationOK.eTypeOutput = E_IO2_Type.NC, gProcess.bSetCaseValidationOK, gProcess.bSetCaseValidationNOK), SEL(gDevice.stMachineConfig.st_Q_CaseValidationOK.eTypeOutput = E_IO2_Type.NC, gProcess.bSetEarlyCaseValidationOK, gProcess.bSetEarlyCaseValidationNOK));
gIOFiltered.stCaseValidationOK.bOutputEnable := _w1;
gProcess.bSetPulseAlarmNOK R= _w1;

// NETWORK 5
fbCaseValidationOK(
    bEnable := gIOFiltered.stCaseValidationOK.bOutputEnable,
    eTypeOutput := gDevice.stMachineConfig.st_Q_CaseValidationOK.eTypeOutput,
    tOutputDelayed := gDevice.stMachineConfig.st_Q_CaseValidationOK.tOutputDelayed,
    tOutputLocked := gDevice.stMachineConfig.st_Q_CaseValidationOK.tOutputLocked,
    bProcessedDelayedOutput => gIOFiltered.stCaseValidationOK.bDelayedOutput,
    bProcessedLockedOutput => gIOFiltered.stCaseValidationOK.bLockedOutput,
    bProcessedDelayedLockedOutput => gIOFiltered.stCaseValidationOK.bDelayedLockedOtput); // FB_IO2_OutputCtrl
gIOFiltered.stCaseValidationOK.bStateOutput := fbCaseValidationOK.bProcessedOutput;

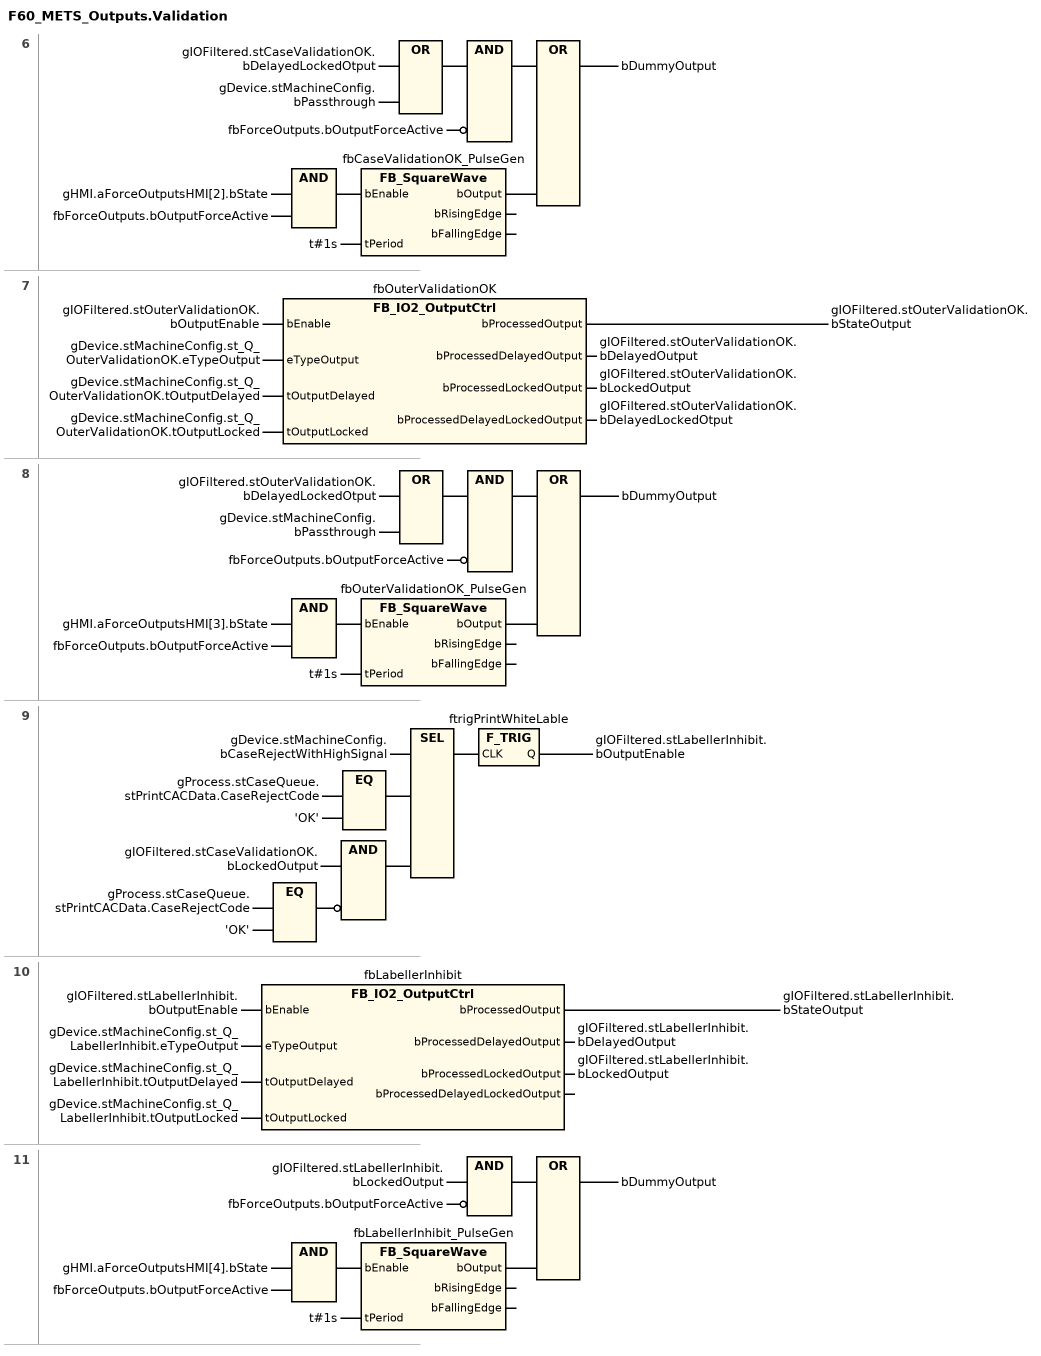
// NETWORK 6
fbCaseValidationOK_PulseGen(bEnable := gHMI.aForceOutputsHMI[2].bState AND fbForceOutputs.bOutputForceActive, tPeriod := t#1s); // FB_SquareWave
bDummyOutput := (gIOFiltered.stCaseValidationOK.bDelayedLockedOtput OR gDevice.stMachineConfig.bPassthrough) AND NOT fbForceOutputs.bOutputForceActive OR fbCaseValidationOK_PulseGen.bOutput;

// NETWORK 7
fbOuterValidationOK(
    bEnable := gIOFiltered.stOuterValidationOK.bOutputEnable,
    eTypeOutput := gDevice.stMachineConfig.st_Q_OuterValidationOK.eTypeOutput,
    tOutputDelayed := gDevice.stMachineConfig.st_Q_OuterValidationOK.tOutputDelayed,
    tOutputLocked := gDevice.stMachineConfig.st_Q_OuterValidationOK.tOutputLocked,
    bProcessedDelayedOutput => gIOFiltered.stOuterValidationOK.bDelayedOutput,
    bProcessedLockedOutput => gIOFiltered.stOuterValidationOK.bLockedOutput,
    bProcessedDelayedLockedOutput => gIOFiltered.stOuterValidationOK.bDelayedLockedOtput); // FB_IO2_OutputCtrl
gIOFiltered.stOuterValidationOK.bStateOutput := fbOuterValidationOK.bProcessedOutput;

// NETWORK 8
fbOuterValidationOK_PulseGen(bEnable := gHMI.aForceOutputsHMI[3].bState AND fbForceOutputs.bOutputForceActive, tPeriod := t#1s); // FB_SquareWave
bDummyOutput := (gIOFiltered.stOuterValidationOK.bDelayedLockedOtput OR gDevice.stMachineConfig.bPassthrough) AND NOT fbForceOutputs.bOutputForceActive OR fbOuterValidationOK_PulseGen.bOutput;

// NETWORK 9
ftrigPrintWhiteLable(CLK := SEL(gDevice.stMachineConfig.bCaseRejectWithHighSignal, gProcess.stCaseQueue.stPrintCACData.CaseRejectCode = 'OK', gIOFiltered.stCaseValidationOK.bLockedOutput AND NOT (gProcess.stCaseQueue.stPrintCACData.CaseRejectCode = 'OK'))); // F_TRIG
gIOFiltered.stLabellerInhibit.bOutputEnable := ftrigPrintWhiteLable.Q;

// NETWORK 10
fbLabellerInhibit(
    bEnable := gIOFiltered.stLabellerInhibit.bOutputEnable,
    eTypeOutput := gDevice.stMachineConfig.st_Q_LabellerInhibit.eTypeOutput,
    tOutputDelayed := gDevice.stMachineConfig.st_Q_LabellerInhibit.tOutputDelayed,
    tOutputLocked := gDevice.stMachineConfig.st_Q_LabellerInhibit.tOutputLocked,
    bProcessedDelayedOutput => gIOFiltered.stLabellerInhibit.bDelayedOutput,
    bProcessedLockedOutput => gIOFiltered.stLabellerInhibit.bLockedOutput); // FB_IO2_OutputCtrl
gIOFiltered.stLabellerInhibit.bStateOutput := fbLabellerInhibit.bProcessedOutput;

// NETWORK 11
fbLabellerInhibit_PulseGen(bEnable := gHMI.aForceOutputsHMI[4].bState AND fbForceOutputs.bOutputForceActive, tPeriod := t#1s); // FB_SquareWave
bDummyOutput := gIOFiltered.stLabellerInhibit.bLockedOutput AND NOT fbForceOutputs.bOutputForceActive OR fbLabellerInhibit_PulseGen.bOutput;
END_ACTION

END_PROGRAM

(* stored: Version 1.1.0.1
   POU F60_METS_Outputs: Id {8b8a37f7-20ef-418a-8b43-14fbd9abc020}, SpecialFunc None
   Action _DT: Id {31ed5904-2822-400b-80c5-7c9e6df7ffa4}
   Action _LogOutputs: Id {27381104-c9c6-4c7b-9703-0972eaede7cb}
   Action AnalogValue: Id {3cd36843-bef7-4dd1-ba5d-cf5877ab9e3e}
   Action Cameras: Id {c58bcaa4-73e1-446f-9da9-f55ab33a2fb5}
   Action CamerasLightning: Id {c23bfd41-7216-4fbf-a5b8-0ca2bc838a76}
   Action CamerasPower: Id {99bd1f6e-fa83-4645-847f-93440ec4b187}
   Action Cylinders: Id {886d1299-d06d-4703-8267-5ae576093e52}
   Action Drives: Id {c4432415-cdfd-4d45-a102-a1885655459d}
   Action Labellers: Id {a3bb7441-4c2d-4a56-bbcc-99595d1413dd}
   Action LightPole: Id {a636e5cc-9a29-4249-a1a1-118369159d7e}
   Action Safety: Id {41d0ba36-a839-4c15-919a-18d5f3e818fd}
   Action SystemRun: Id {613754eb-79b7-45de-b07d-d8645c561a9e}
   Action Validation: Id {d64a37c6-9688-4899-81fa-42f1e833d026} *)
